(* CODESYS project integratedManufacturingSystem.export

Project tree, tasks and I/O mapping:
  Device : CODESYS Control Win V3 x64, CODESYS, version 3.5.22.30
    application Application
      libraries: Standard, 3.5.22.0 (System)
      task MainTask (cyclic, interval t#20ms, priority 1) calls PLC_PRG
      DUTs/
        data type E_AssemblerState
        data type E_BatchStorageState
        data type E_MachiningCellState
        data type E_PackoutCarrierState
        data type E_PackoutLoaderState
        data type E_PackoutState
        data type E_PairCoordinatorState
        data type E_PairDiverterState
        data type E_PlantState
        data type E_ProductionPhase
        data type E_RackSlotState
        data type E_StorageState
        data type E_TankState
        data type E_TransferState
      GVLs/
        global variables FIO
        global variables PlantConstants
        global variables SCADA
      POUs/
        function block FB_AssemblerCell [ST]
        function block FB_AssemblyUnit [ST]
        function block FB_BatchStorageUnit [ST]
        function block FB_MachiningCell [ST]
        function block FB_MasterOperatorControl [ST]
        function block FB_PackoutCarrierStation [ST]
        function block FB_PackoutLoader [ST]
        function block FB_PairDiverter [ST]
        function block FB_PlantCoordinator [ST]
        function block FB_RackManager [ST]
        function block FB_Storage [ST]
        function block FB_Tank [ST]
        function block FB_TransferCoordinator [ST]
        function block FB_TwinCellUnit [ST]
        function block FB_UnitOperatorControl [ST]
      program PLC_PRG [ST]
      Symbols
*)

// Device/Application/DUTs/E_AssemblerState
{attribute 'qualified_only'}
{attribute 'strict'}
TYPE E_AssemblerState :
(
    Stopped               := 0,
    Homing                := 10,
    WaitingForParts       := 20,
    ClampingParts         := 30,
    LoweringToLid         := 40,
    GrippingLid           := 50,
    ReleasingLidClamp     := 60,
    RaisingLid            := 70,
    MovingToBase          := 80,
    LoweringToBase        := 90,
    ReleasingLid          := 100,
    RaisingFromBase       := 110,
    ReturningHome         := 120,
    ReleasingProduct      := 130,
    WaitingForProductExit := 140,
    Faulted               := 900
);
END_TYPE

// Device/Application/DUTs/E_BatchStorageState
{attribute 'qualified_only'}
{attribute 'strict'}
TYPE E_BatchStorageState :
(
    Stopped                   := 0,
    Idle                      := 10,
    ReservingSlot             := 20,
    WaitingForBatch           := 30,
    DischargingBatch          := 40,
    StoringProduct            := 50,
    CommittingInventory       := 60,
    WaitingForStorageComplete := 70,
    Faulted                   := 900
);
END_TYPE

// Device/Application/DUTs/E_MachiningCellState
{attribute 'qualified_only'}
{attribute 'strict'}
TYPE E_MachiningCellState :
(
    Stopped          := 0,
    Ready            := 10,
    FeedingRaw       := 20,
    WaitingForPickup := 30,
    Processing       := 40,
    Complete         := 50,
    Faulted          := 900
);
END_TYPE

// Device/Application/DUTs/E_PackoutCarrierState
{attribute 'qualified_only'}
{attribute 'strict'}
TYPE E_PackoutCarrierState :
(
    Stopped                      := 0,
    WaitingForCarrierRequest     := 10,
    FeedingCarrier               := 20,
    HoldingCarrierAtLoad         := 30,
    RequestingPlantStorage       := 40,
    TransferringCarrier          := 50,
    WaitingForDownstreamAckClear := 60,
    Faulted                      := 900
);
END_TYPE

// Device/Application/DUTs/E_PackoutLoaderState
{attribute 'qualified_only'}
{attribute 'strict'}
TYPE E_PackoutLoaderState :
(
    Stopped                  := 0,
    Homing                   := 10,
    WaitingForCarrier        := 20,
    WaitingForProduct        := 30,
    MovingToProduct          := 35,
    LoweringToProduct        := 40,
    GrippingProduct          := 50,
    RaisingProduct           := 60,
    MovingToCarrier          := 70,
    LoweringToCarrier        := 80,
    ReleasingProduct         := 90,
    RaisingFromCarrier       := 100,
    ReturningHome            := 110,
    VerifyingLoad            := 120,
    WaitingForLoadAcceptance := 130,
    Complete                 := 140,
    Faulted                  := 900
);
END_TYPE

// Device/Application/DUTs/E_PackoutState
{attribute 'qualified_only'}
{attribute 'strict'}
TYPE E_PackoutState :
(
    Stopped            := 0,
    Homing             := 10,
    WaitingForProduct  := 20,
    RequestingCarrier  := 30,
    PositioningCarrier := 40,
    LoweringToProduct  := 50,
    GrippingProduct    := 60,
    RaisingProduct     := 70,
    MovingToCarrier    := 80,
    LoweringToCarrier  := 90,
    ReleasingProduct   := 100,
    RaisingFromCarrier := 110,
    ReturningHome      := 120,
    VerifyingLoad      := 130,
    ReleasingCarrier   := 140,
    Complete           := 150,
    Faulted            := 900
);
END_TYPE

// Device/Application/DUTs/E_PairCoordinatorState
{attribute 'qualified_only'}
{attribute 'strict'}
TYPE E_PairCoordinatorState :
(
    Stopped          := 0,
    Ready            := 10,
    WaitPairComplete := 20,
    MergeClearance   := 30,
    Faulted          := 900
);
END_TYPE

// Device/Application/DUTs/E_PairDiverterState
{attribute 'qualified_only'}
{attribute 'strict'}
TYPE E_PairDiverterState :
(
    Idle                    := 0,
    ReleasingBase           := 10,
    ReleasingLid            := 20,
    PassingBase             := 30,
    WaitingForLidAtPusher   := 40,
    PositioningLid          := 50,
    PushingLid              := 60,
    WaitingForPartsAtPlace  := 70,
    Complete                := 80,
    Faulted                 := 900
);
END_TYPE

// Device/Application/DUTs/E_PlantState
{attribute 'qualified_only'}
{attribute 'strict'}
TYPE E_PlantState :
(
    Stopped          := 0,
    Ready            := 10,
    Starting         := 20,
    Running          := 30,
    Stopping         := 40,
    Faulted          := 900,
    RecoveryRequired := 910
);
END_TYPE

// Device/Application/DUTs/E_ProductionPhase
{attribute 'qualified_only'}
{attribute 'strict'}
TYPE E_ProductionPhase :
(
    Idle              := 0,
    ReservingStorage  := 10,
    ProducingPair     := 20,
    Assembling        := 30,
    WaitingForPackout := 40,
    Batching          := 50,
    Storing           := 60,
    Complete          := 70
);
END_TYPE

// Device/Application/DUTs/E_RackSlotState
{attribute 'qualified_only'}
{attribute 'strict'}
TYPE E_RackSlotState :
(
    Free     := 0,
    Reserved := 10,
    Occupied := 20,
    Unknown  := 900
);
END_TYPE

// Device/Application/DUTs/E_StorageState
{attribute 'qualified_only'}
{attribute 'strict'}
TYPE E_StorageState :
(
    Stopped                := 0,
    Idle                   := 10,
    ReceivingProduct       := 20,
    ExtendingToLoad        := 30,
    LiftingProduct         := 40,
    RetractingWithProduct  := 50,
    MovingToRack           := 60,
    ExtendingToRack        := 70,
    LoweringProduct        := 80,
    RetractingAfterDeposit := 90,
    ReturningHome          := 100,
    Complete               := 110,
    Faulted                := 900
);
END_TYPE

// Device/Application/DUTs/E_TankState
{attribute 'qualified_only'}
{attribute 'strict'}
TYPE E_TankState :
(
    Stopped     := 0,
    Idle        := 10,
    Filling     := 20,
    BatchReady  := 30,
    Discharging := 40,
    Faulted     := 900
);
END_TYPE

// Device/Application/DUTs/E_TransferState
{attribute 'qualified_only'}
{attribute 'strict'}
TYPE E_TransferState :
(
    Idle                   := 0,
    WaitingForReady        := 10,
    Transferring           := 20,
    WaitingForRequestClear := 30,
    Faulted                := 900
);
END_TYPE

// Device/Application/GVLs/FIO
{attribute 'qualified_only'}
VAR_GLOBAL
    // Factory I/O lifecycle
    rFactoryIOTimeScale : REAL;
    xFactoryIOPaused    : BOOL;
    xFactoryIOReset     : BOOL;
    xFactoryIORunning   : BOOL;
	
	// MASTER operator panel
	xMasterAutoModeSelected       : BOOL;
	xMasterEmergencyStopHealthy   : BOOL;
	xMasterManualModeSelected     : BOOL;
	xMasterResetLightCmd          : BOOL;
	xMasterResetPB                : BOOL;
	xMasterStackGreenCmd          : BOOL;
	xMasterStackRedCmd            : BOOL;
	xMasterStackYellowCmd         : BOOL;
	xMasterStartLightCmd          : BOOL;
	xMasterStartPB                : BOOL;
	xMasterStopCircuitHealthy     : BOOL;
	xMasterStopLightCmd           : BOOL;

    // Plant panel
    xPlantAutoModeSelected     : BOOL;
    xPlantEmergencyStopHealthy : BOOL;
    xPlantManualModeSelected   : BOOL;
    xPlantResetPB              : BOOL;
    xPlantStartPB              : BOOL;
    xPlantStopCircuitHealthy   : BOOL;

    // Twin Cell
    diTwinCellBasesCenterProgress : DINT;
    diTwinCellLidsCenterProgress  : DINT;
    xTwinCellBasesCenterBusy      : BOOL;
    xTwinCellBasesCenterHasError  : BOOL;
    xTwinCellBasesCenterOpened    : BOOL;
    xTwinCellBasesEntryBeamClear  : BOOL;
    xTwinCellBasesExitBeamClear   : BOOL;
    xTwinCellEmergencyStopHealthy : BOOL;
    xTwinCellLidsCenterBusy       : BOOL;
    xTwinCellLidsCenterHasError   : BOOL;
    xTwinCellLidsCenterOpened     : BOOL;
    xTwinCellLidsEntryBeamClear   : BOOL;
    xTwinCellLidsExitBeamClear    : BOOL;
    xTwinCellLocalModeSelected    : BOOL;
    xTwinCellPlantModeSelected    : BOOL;
    xTwinCellResetPB              : BOOL;
    xTwinCellStartPB              : BOOL;
    xTwinCellStopCircuitHealthy   : BOOL;

    // Pair sorter
    xPairSorterCountBeamClear  : BOOL;
    xPairSorterPusherAtBack    : BOOL;
    xPairSorterPusherAtFront   : BOOL;
    xPairSorterPusherBeamClear : BOOL;

    // Assembly
    xAssemblyBaseAtPlace            : BOOL;
    xAssemblyBaseClamped            : BOOL;
    xAssemblyBasesPositionerAtLimit : BOOL;
    xAssemblyItemDetected           : BOOL;
    xAssemblyLidAtPlace             : BOOL;
    xAssemblyLidClamped             : BOOL;
    xAssemblyLidsPositionerAtLimit  : BOOL;
    xAssemblyMovingX                : BOOL;
    xAssemblyMovingZ                : BOOL;
    xAssemblyProductAtOutfeed       : BOOL;

    // Packout
    xPackoutItemDetected           : BOOL;
    xPackoutMovingX                : BOOL;
    xPackoutMovingZ                : BOOL;
    xPackoutPalletAtLoadBeamClear  : BOOL;
    xPackoutProductAtPickBeamClear : BOOL;
    xPackoutProductLoaded          : BOOL;

    // Tank and transfer
    rTankFlowV         : REAL;
    rTankLevelV        : REAL;
    xTankCarrierAtFill : BOOL;
    xTankLevelHighHigh : BOOL;

    // Storage and rack
    xStorageAtEntryBeamClear  : BOOL;
    xStorageAtExitBeamClear   : BOOL;
    xStorageAtUnloadBeamClear : BOOL;
    xStorageForkAtLeft        : BOOL;
    xStorageForkAtMiddle      : BOOL;
    xStorageForkAtRight       : BOOL;
    xStorageLoadBeamClear     : BOOL;
    xStorageMovingX           : BOOL;
    xStorageMovingZ           : BOOL;
	
    // Factory I/O lifecycle — PLC to Factory I/O
    diFactoryIOCameraPositionCmd : DINT;
    xFactoryIOPauseCmd           : BOOL;
    xFactoryIOResetCmd           : BOOL;
    xFactoryIORunCmd             : BOOL;

    // Plant panel — PLC to Factory I/O
    xPlantResetLightCmd : BOOL;
    xPlantStartLightCmd : BOOL;
    xPlantStopLightCmd  : BOOL;

    // Twin Cell — PLC to Factory I/O
    diTwinCellBasesCellCounterDisplay  : DINT;
    diTwinCellBasesPanelCounterDisplay : DINT;
    diTwinCellLidsCellCounterDisplay   : DINT;
    diTwinCellLidsPanelCounterDisplay  : DINT;
    xTwinCellBasesCenterProduceCmd     : BOOL;
    xTwinCellBasesCenterResetCmd       : BOOL;
    xTwinCellBasesCenterStartCmd       : BOOL;
    xTwinCellBasesCenterStopCmd        : BOOL;
    xTwinCellBasesEmitterCmd           : BOOL;
    xTwinCellBasesExitConveyor1Cmd     : BOOL;
    xTwinCellBasesExitConveyor2Cmd     : BOOL;
    xTwinCellBasesRawConveyorCmd       : BOOL;
    xTwinCellLidsCenterProduceCmd      : BOOL;
    xTwinCellLidsCenterResetCmd        : BOOL;
    xTwinCellLidsCenterStartCmd        : BOOL;
    xTwinCellLidsCenterStopCmd         : BOOL;
    xTwinCellLidsEmitterCmd            : BOOL;
    xTwinCellLidsExitConveyor1Cmd      : BOOL;
    xTwinCellLidsExitConveyor2Cmd      : BOOL;
    xTwinCellLidsRawConveyorCmd        : BOOL;
    xTwinCellResetLightCmd             : BOOL;
    xTwinCellStartLightCmd             : BOOL;
    xTwinCellStopLightCmd              : BOOL;

    // Pair sorter — PLC to Factory I/O
    diPairSorterDetectionCountDisplay : DINT;
    xPairSorterBaseCurveConveyorCmd   : BOOL;
    xPairSorterInfeedConveyorCmd      : BOOL;
    xPairSorterPusherCmd              : BOOL;
    xPairSorterPusherZoneConveyorCmd  : BOOL;

    // Assembly — PLC to Factory I/O
    xAssemblyBaseClampCmd            : BOOL;
    xAssemblyBasesConveyorCmd        : BOOL;
    xAssemblyBasesPositionerRaiseCmd : BOOL;
    xAssemblyGrabCmd                 : BOOL;
    xAssemblyLidClampCmd             : BOOL;
    xAssemblyLidsConveyorCmd         : BOOL;
    xAssemblyLidsPositionerRaiseCmd  : BOOL;
    xAssemblyMoveXCmd                : BOOL;
    xAssemblyMoveZCmd                : BOOL;

    // Packout — PLC to Factory I/O
    xPackoutBufferConveyor1Cmd       : BOOL;
    xPackoutBufferConveyor2Cmd       : BOOL;
    xPackoutBufferConveyor3Cmd       : BOOL;
    xPackoutCarrierConveyorCmd       : BOOL;
    xPackoutCarrierEmitterCmd        : BOOL;
    xPackoutCarrierInfeedConveyorCmd : BOOL;
    xPackoutGrabCmd                  : BOOL;
    xPackoutMoveXCmd                 : BOOL;
    xPackoutMoveZCmd                 : BOOL;
    xPackoutPickConveyorCmd          : BOOL;

    // Tank and transfer — PLC to Factory I/O
    rTankDischargeValveCmdV   : REAL;
    rTankFillValveCmdV        : REAL;
    xTankTransferConveyor1Cmd : BOOL;
    xTankTransferConveyor2Cmd : BOOL;
    xTankTransferConveyor3Cmd : BOOL;
    xTankTransferConveyor4Cmd : BOOL;

    // Storage and rack — PLC to Factory I/O
    wStorageTargetPositionCmd : WORD := 55;
    xStorageEntryConveyorCmd  : BOOL;
    xStorageExitConveyorCmd   : BOOL;
    xStorageExitRemoverCmd    : BOOL;
    xStorageForksLeftCmd      : BOOL;
    xStorageForksRightCmd     : BOOL;
    xStorageLiftCmd           : BOOL;
    xStorageLoadConveyorCmd   : BOOL;
    xStorageUnloadConveyorCmd : BOOL;

    // Stack lights — PLC to Factory I/O
    xPackoutStackGreenCmd  : BOOL;
    xPackoutStackRedCmd    : BOOL;
    xPackoutStackYellowCmd : BOOL;
    xPlantStackGreenCmd    : BOOL;
    xPlantStackRedCmd      : BOOL;
    xPlantStackYellowCmd   : BOOL;
    xStorageStackGreenCmd  : BOOL;
    xStorageStackRedCmd    : BOOL;
    xStorageStackYellowCmd : BOOL;
    xTankStackGreenCmd     : BOOL;
    xTankStackRedCmd       : BOOL;
    xTankStackYellowCmd    : BOOL;
END_VAR

// Device/Application/GVLs/PlantConstants
{attribute 'qualified_only'}
VAR_GLOBAL CONSTANT
    tPairTransferTimeout    : TIME := T#2M;
    tProductTransferTimeout : TIME := T#30S;
    wStorageHomePosition    : WORD := 55;
END_VAR

// Device/Application/GVLs/SCADA
{attribute 'symbol' := 'read'}
{attribute 'qualified_only'}
VAR_GLOBAL
    // Ignition to PLC — momentary requests
	 {attribute 'symbol' := 'readwrite'}
    xResetReq : BOOL;
	 {attribute 'symbol' := 'readwrite'}
    xStartReq : BOOL;
	 {attribute 'symbol' := 'readwrite'}
    xStopReq  : BOOL;
	 {attribute 'symbol' := 'readwrite'}
	xAutoModeSelected 		  : BOOL := FALSE;

    // PLC to Ignition — plant
    diPlantCompletedLoadCount : DINT;
    ePlantState               : E_PlantState := E_PlantState.Stopped;
    eProductionPhase          : E_ProductionPhase := E_ProductionPhase.Idle;
    uiPlantFaultCode          : UINT;
	xAllEmergencyStopsHealthy : BOOL;
	xAutoModeActive           : BOOL;
	xFactoryIORunning         : BOOL;
	xManualModeActive         : BOOL;
    xPlantFaulted             : BOOL;
    xPlantRecoveryRequired    : BOOL;
    xPlantRunning             : BOOL;
    xPlantStopPending         : BOOL;

    // PLC to Ignition — Twin Cell
    diTwinCellPairCount : DINT;
    uiTwinCellFaultCode : UINT;
    xTwinCellBusy       : BOOL;
    xTwinCellFaulted    : BOOL;
    xTwinCellReady      : BOOL;

    // PLC to Ignition — pair transfer
    ePairTransferState       : E_TransferState := E_TransferState.Idle;
    uiPairTransferFaultCode  : UINT;
    xPairTransferAck         : BOOL;
    xPairTransferFaulted     : BOOL;
    xPairTransferPermit      : BOOL;
    xPairTransferReady       : BOOL;
    xPairTransferReq         : BOOL;

    // PLC to Ignition — pair sorter
    diPairSorterDetectionCount : DINT;
    ePairDiverterState         : E_PairDiverterState := E_PairDiverterState.Idle;
    uiPairSorterFaultCode      : UINT;
    xPairSorterFaulted         : BOOL;
    xPairSorterPartAtPusher    : BOOL;

    // PLC to Ignition — assembly
    diAssemblyProductCount : DINT;
    eAssemblyState         : E_AssemblerState := E_AssemblerState.Stopped;
    uiAssemblyFaultCode    : UINT;
    xAssemblyBusy          : BOOL;
    xAssemblyFaulted       : BOOL;
    xAssemblyReady         : BOOL;

    // PLC to Ignition — product transfer
    eProductTransferState      : E_TransferState := E_TransferState.Idle;
    uiProductTransferFaultCode : UINT;
    xProductTransferAck        : BOOL;
    xProductTransferFaulted    : BOOL;
    xProductTransferPermit     : BOOL;
    xProductTransferReady      : BOOL;
    xProductTransferReq        : BOOL;

    // PLC to Ignition — packout
	diPackoutProductCount        : DINT;
	
	ePackoutCarrierState         : E_PackoutCarrierState :=
									   E_PackoutCarrierState.Stopped;
	ePackoutLoaderState          : E_PackoutLoaderState :=
									   E_PackoutLoaderState.Stopped;
	
	uiPackoutCarrierFaultCode    : UINT;
	uiPackoutLoaderFaultCode     : UINT;
	
	xPackoutBusy                 : BOOL;
	xPackoutCarrierBusy          : BOOL;
	xPackoutCarrierFaulted       : BOOL;
	xPackoutCarrierReady         : BOOL;
	xPackoutFaulted              : BOOL;
	xPackoutLoaderBusy           : BOOL;
	xPackoutLoaderFaulted        : BOOL;
	xPackoutLoaderReady          : BOOL;
	xPackoutReady                : BOOL;

    // PLC to Ignition — process and storage
    eBatchStorageState       : E_BatchStorageState := E_BatchStorageState.Stopped;
    eStorageState            : E_StorageState := E_StorageState.Stopped;
    eTankState               : E_TankState := E_TankState.Stopped;
    rTankLevelPct            : REAL;
    uiRackFreeCount          : UINT;
    uiRackOccupiedCount      : UINT;
    uiRackReservedCount      : UINT;
    uiRackUnknownCount       : UINT;
    uiStorageFaultCode       : UINT;
    wStorageReservedPosition : WORD;
    xPackoutPalletAtLoad     : BOOL;
    xPackoutProductAtPick    : BOOL;
    xPackoutProductLoaded    : BOOL;
    xRackFull                : BOOL;
    xStorageBusy             : BOOL;
    xStorageFaulted          : BOOL;
    xStorageReady            : BOOL;
	
	// Maintained automatic-mode request from Ignition.
	{attribute 'symbol' := 'readwrite'}
	xIgnitionAutoModeReq : BOOL;
END_VAR

// Device/Application/PLC_PRG
PROGRAM PLC_PRG
VAR
    // Function-block instances
	fbAssemblyUnit                  : FB_AssemblyUnit;
	fbBatchStorageOperatorControl   : FB_UnitOperatorControl;
	fbBatchStorageUnit              : FB_BatchStorageUnit;
	fbMasterOperatorControl         : FB_MasterOperatorControl;
	fbPackoutCarrierStation         : FB_PackoutCarrierStation;
	fbPackoutLoader                 : FB_PackoutLoader;
	fbPairDiverter                  : FB_PairDiverter;
	fbPairTransfer                  : FB_TransferCoordinator;
	fbPlantCoordinator              : FB_PlantCoordinator;
	fbProductTransfer               : FB_TransferCoordinator;
	fbTwinCellOperatorControl       : FB_UnitOperatorControl;
	fbTwinCellUnit                  : FB_TwinCellUnit;

    // Normalised physical inputs
    rTankLevelPct               : REAL;
	xBatchStorageTransferActive : BOOL;
    xPackoutPalletAtLoad        : BOOL;
    xPackoutProductAtPick       : BOOL;
    xPairSorterCountDetected    : BOOL;
    xPairSorterPartAtPusher     : BOOL;
    xStorageAtEntry             : BOOL;
    xStorageAtExit              : BOOL;
    xStorageAtUnload            : BOOL;
	xStorageCraneAtHome         : BOOL;
    xStorageProductAtLoad       : BOOL;
    xTwinCellBasesEntryDetected : BOOL;
    xTwinCellBasesExitDetected  : BOOL;
    xTwinCellLidsEntryDetected  : BOOL;
    xTwinCellLidsExitDetected   : BOOL;
	xTwinCellOutputPermit 		: BOOL := TRUE;

    // Safety and commissioning
    xAllEmergencyStopsHealthy : BOOL;
	xAnyFault              	  : BOOL;
	xOutputPermit             : BOOL;
	xPairSorterOutputPermit   : BOOL := TRUE;
    xPairTransferActive    	  : BOOL;
    xProductTransferActive    : BOOL;
	xStorageOutputPermit      : BOOL;
END_VAR

// =============================================================
// 1. INPUT IMAGE AND POLARITY NORMALISATION
// =============================================================
rTankLevelPct := FIO.rTankLevelV * 10.0;

xPackoutPalletAtLoad := NOT FIO.xPackoutPalletAtLoadBeamClear;
xPackoutProductAtPick := NOT FIO.xPackoutProductAtPickBeamClear;
xPairSorterCountDetected := NOT FIO.xPairSorterCountBeamClear;
xPairSorterPartAtPusher := NOT FIO.xPairSorterPusherBeamClear;

xStorageAtEntry := NOT FIO.xStorageAtEntryBeamClear;
xStorageAtExit := NOT FIO.xStorageAtExitBeamClear;
xStorageAtUnload := NOT FIO.xStorageAtUnloadBeamClear;
xStorageCraneAtHome :=
    (FIO.wStorageTargetPositionCmd =
        PlantConstants.wStorageHomePosition)
    AND FIO.xStorageForkAtMiddle
    AND NOT FIO.xStorageMovingX
    AND NOT FIO.xStorageMovingZ;
xStorageProductAtLoad := NOT FIO.xStorageLoadBeamClear;

xTwinCellBasesEntryDetected := NOT FIO.xTwinCellBasesEntryBeamClear;
xTwinCellBasesExitDetected := NOT FIO.xTwinCellBasesExitBeamClear;
xTwinCellLidsEntryDetected := NOT FIO.xTwinCellLidsEntryBeamClear;
xTwinCellLidsExitDetected := NOT FIO.xTwinCellLidsExitBeamClear;

// =============================================================
// 2. SAFETY AND COMMISSIONING CONDITIONS
// =============================================================
xAllEmergencyStopsHealthy :=
    FIO.xMasterEmergencyStopHealthy
	AND FIO.xPlantEmergencyStopHealthy
    AND FIO.xTwinCellEmergencyStopHealthy;

// Global commissioned outputs are permitted.
// Uncommissioned zones remain protected by their individual permits.
xOutputPermit := TRUE;

// =============================================================
// 3. OPERATOR CONTROL
// =============================================================
fbMasterOperatorControl(
    xAutoModeSelected :=
		FIO.xMasterAutoModeSelected
		OR SCADA.xIgnitionAutoModeReq,
    xEmergencyStopHealthy := xAllEmergencyStopsHealthy,
    xFactoryIORunning := FIO.xFactoryIORunning,
    xManualModeSelected := FIO.xMasterManualModeSelected,
    xPlantFaulted := fbPlantCoordinator.xFaulted,
    xResetPB := FIO.xMasterResetPB OR SCADA.xResetReq,
    xStartPB := FIO.xMasterStartPB OR SCADA.xStartReq,
    xStopCircuitHealthy :=
        FIO.xMasterStopCircuitHealthy
        AND NOT SCADA.xStopReq
);

xBatchStorageTransferActive :=
    fbBatchStorageUnit.xBusy
    OR fbPackoutCarrierStation.xBusy
    OR fbPackoutCarrierStation.xLoadedCarrierReq
    OR fbPackoutLoader.xBusy
    OR fbPackoutLoader.xLoadComplete;

fbBatchStorageOperatorControl(
    xEmergencyStopHealthy := xAllEmergencyStopsHealthy,
    xLocalModeSelected := FIO.xPlantManualModeSelected,
    xLocalResetPB := FIO.xPlantResetPB,
    xLocalStartPB := FIO.xPlantStartPB,
    xLocalStopHealthy := FIO.xPlantStopCircuitHealthy,
    xMasterAutoModeActive :=
        fbMasterOperatorControl.xAutoModeActive,
    xMasterEnable := fbMasterOperatorControl.xEnable,
    xMasterManualModeActive :=
        fbMasterOperatorControl.xManualModeActive,
    xMasterModeSelected := FIO.xPlantAutoModeSelected,
    xMasterResetPulse := fbMasterOperatorControl.xResetPulse,
    xMasterRun := fbPlantCoordinator.xRunning,
    xTransferActive := xBatchStorageTransferActive
);

xPairTransferActive :=
    fbPairTransfer.eState <> E_TransferState.Idle;

xProductTransferActive :=
    (fbProductTransfer.eState <> E_TransferState.Idle)
    OR fbPackoutLoader.xBusy
    OR fbPackoutLoader.xLoadComplete;

fbTwinCellOperatorControl(
    xEmergencyStopHealthy := xAllEmergencyStopsHealthy,
    xLocalModeSelected := FIO.xTwinCellLocalModeSelected,
    xLocalResetPB := FIO.xTwinCellResetPB,
    xLocalStartPB := FIO.xTwinCellStartPB,
    xLocalStopHealthy := FIO.xTwinCellStopCircuitHealthy,
	xMasterAutoModeActive :=
    	fbMasterOperatorControl.xAutoModeActive,
    xMasterEnable := fbMasterOperatorControl.xEnable,
	xMasterManualModeActive :=
    	fbMasterOperatorControl.xManualModeActive,
    xMasterModeSelected := FIO.xTwinCellPlantModeSelected,
    xMasterResetPulse := fbMasterOperatorControl.xResetPulse,
    xMasterRun := fbPlantCoordinator.xRunning,
    xTransferActive :=
        xPairTransferActive OR xProductTransferActive
);

// =============================================================
// 4. UNIT BOUNDARIES
// =============================================================
fbTwinCellUnit(
    xEnable := fbTwinCellOperatorControl.xEnable,
    xPairAccepted := fbAssemblyUnit.xPairAck,
	xProductionRequest :=
		fbMasterOperatorControl.xAutoRun
		AND fbPlantCoordinator.xAllowNewPair,
    xReset := fbTwinCellOperatorControl.xResetPulse,
    xRun :=
		fbTwinCellOperatorControl.xRun
		AND xTwinCellOutputPermit,
    xTwinCellBasesCenterBusy :=
        FIO.xTwinCellBasesCenterBusy,
    xTwinCellBasesCenterHasError :=
        FIO.xTwinCellBasesCenterHasError,
    xTwinCellBasesCenterOpened :=
        FIO.xTwinCellBasesCenterOpened,
    xTwinCellBasesEntryDetected :=
        xTwinCellBasesEntryDetected,
    xTwinCellBasesExitDetected :=
        xTwinCellBasesExitDetected,
    xTwinCellLidsCenterBusy :=
        FIO.xTwinCellLidsCenterBusy,
    xTwinCellLidsCenterHasError :=
        FIO.xTwinCellLidsCenterHasError,
    xTwinCellLidsCenterOpened :=
        FIO.xTwinCellLidsCenterOpened,
    xTwinCellLidsEntryDetected :=
        xTwinCellLidsEntryDetected,
    xTwinCellLidsExitDetected :=
        xTwinCellLidsExitDetected
);

fbAssemblyUnit(
    xBaseAtPlace :=
        FIO.xAssemblyBaseAtPlace,

    xBaseClamped :=
        FIO.xAssemblyBaseClamped,

    xBasesPositionerAtLimit :=
        FIO.xAssemblyBasesPositionerAtLimit,

    xEnable :=
        fbTwinCellOperatorControl.xEnable
        AND FIO.xFactoryIORunning
        AND xOutputPermit,

    xItemDetected :=
        FIO.xAssemblyItemDetected,

    xLidAtPlace :=
        FIO.xAssemblyLidAtPlace,

    xLidClamped :=
        FIO.xAssemblyLidClamped,

    xMovingX :=
        FIO.xAssemblyMovingX,

    xMovingZ :=
        FIO.xAssemblyMovingZ,

    xProductAtOutfeed :=
        FIO.xAssemblyProductAtOutfeed,

    xProductTransferAck :=
        fbPackoutLoader.xProductTransferAck,

    xReset :=
        fbTwinCellOperatorControl.xResetPulse,

    xRun :=
        fbTwinCellOperatorControl.xRun
);

// =============================================================
// 5. P10-TO-P11 TRANSFER
// =============================================================
fbPairTransfer(
    tTransferTimeout := PlantConstants.tPairTransferTimeout,
    xAck := fbAssemblyUnit.xPairAck,
    xEnable :=
		fbPlantCoordinator.xPairTransferEnable
		AND xPairSorterOutputPermit,
    xReady := fbAssemblyUnit.xPairReady,
    xReq := fbTwinCellUnit.xPairReq,
    xReset := fbMasterOperatorControl.xResetPulse,
	xRun := fbTwinCellOperatorControl.xRun
);

fbPairDiverter(
	tLidPositionTime := T#700MS,
    tStepTimeout := T#45S,
    xAssemblyBaseAtPlace := FIO.xAssemblyBaseAtPlace,
    xAssemblyLidAtPlace := FIO.xAssemblyLidAtPlace,
    xCountDetected := xPairSorterCountDetected,
    xEnable :=
		xAllEmergencyStopsHealthy
		AND FIO.xFactoryIORunning
		AND xOutputPermit
		AND xPairSorterOutputPermit,
		xPartAtPusher := xPairSorterPartAtPusher,
    xPusherAtBack := FIO.xPairSorterPusherAtBack,
    xPusherAtFront := FIO.xPairSorterPusherAtFront,
    xReset := fbMasterOperatorControl.xResetPulse,
	xRun := fbTwinCellOperatorControl.xRun,
	xTransferPermit := fbPairTransfer.xPermit
);

// =============================================================
// 6. P11-TO-PACKOUT LOADER TRANSFER
// =============================================================
fbProductTransfer(
    tTransferTimeout := PlantConstants.tProductTransferTimeout,
    xAck := fbPackoutLoader.xProductTransferAck,
    xEnable := fbPlantCoordinator.xProductTransferEnable,
    xReady := fbPackoutLoader.xProductTransferReady,
    xReq := fbAssemblyUnit.xProductReq,
    xReset := fbMasterOperatorControl.xResetPulse,
	xRun := fbTwinCellOperatorControl.xRun	
);

fbPackoutLoader(
    tStepTimeout := T#20S,
    xCarrierReady := fbPackoutCarrierStation.xCarrierReady,
    xEnable :=
        xAllEmergencyStopsHealthy
		AND FIO.xFactoryIORunning
		AND xOutputPermit,
    xItemDetected := FIO.xPackoutItemDetected,
    xLoadAccepted := fbPackoutCarrierStation.xLoadAccepted,
    xMovingX := FIO.xPackoutMovingX,
    xMovingZ := FIO.xPackoutMovingZ,
    xProductAtPick := xPackoutProductAtPick,
    xProductLoaded := FIO.xPackoutProductLoaded,
    xProductTransferPermit := fbProductTransfer.xPermit,
    xReset := fbTwinCellOperatorControl.xResetPulse,
	xRun :=
		fbTwinCellOperatorControl.xRun
		AND fbPlantCoordinator.xRunning
);

fbPackoutCarrierStation(
    tStepTimeout := T#30S,
    xCarrierReq := fbPackoutLoader.xCarrierReq,
    xDownstreamAck := fbBatchStorageUnit.xProductTransferAck,
    xDownstreamReady := fbBatchStorageUnit.xProductTransferReady,
    xEnable :=
        fbBatchStorageOperatorControl.xEnable
        AND FIO.xFactoryIORunning
        AND xOutputPermit,
    xLoadComplete := fbPackoutLoader.xLoadComplete,
    xPalletAtLoad := xPackoutPalletAtLoad,
    xProductLoaded := FIO.xPackoutProductLoaded,
    xReset := fbBatchStorageOperatorControl.xResetPulse,
    xRun :=
        fbBatchStorageOperatorControl.xRun
        AND fbPlantCoordinator.xRunning
);

// =============================================================
// 7. PACKOUT-TO-PLANT STORAGE BOUNDARY
// =============================================================
fbBatchStorageUnit(
    rTankLevelV := FIO.rTankLevelV,
	wStorageHomePosition :=
        PlantConstants.wStorageHomePosition,
    xEnable := fbBatchStorageOperatorControl.xEnable,
    xPackoutPalletAtLoad := xPackoutPalletAtLoad,
    xPackoutProductLoaded := FIO.xPackoutProductLoaded,
    xProductTransferReq :=
        fbPackoutCarrierStation.xLoadedCarrierReq,
    xReset := fbBatchStorageOperatorControl.xResetPulse,
    xRun := fbBatchStorageOperatorControl.xRun,
    xStorageAtEntry := xStorageAtEntry,
	 xStorageCraneAtHome := xStorageCraneAtHome,
    xStorageForkAtLeft := FIO.xStorageForkAtLeft,
    xStorageForkAtMiddle := FIO.xStorageForkAtMiddle,
    xStorageForkAtRight := FIO.xStorageForkAtRight,
    xStorageMovingX := FIO.xStorageMovingX,
    xStorageMovingZ := FIO.xStorageMovingZ,
    xStorageProductAtLoad := xStorageProductAtLoad,
    xTankCarrierAtFill := FIO.xTankCarrierAtFill,
    xTankLevelHighHigh := FIO.xTankLevelHighHigh
);

// =============================================================
// 8. PLANT COORDINATION
// =============================================================
xAnyFault :=
    fbAssemblyUnit.xFaulted
    OR fbBatchStorageUnit.xFaulted
    OR fbPackoutCarrierStation.xFaulted
    OR fbPackoutLoader.xFaulted
    OR fbPairDiverter.xFaulted
    OR fbPairTransfer.xFaulted
    OR fbProductTransfer.xFaulted
    OR fbTwinCellUnit.xFaulted;

fbPlantCoordinator(
    xAnyFault := xAnyFault,
    xAutoRun := fbMasterOperatorControl.xAutoRun,
    xBatchStorageReady := fbBatchStorageUnit.xReady,
    xEnable := fbMasterOperatorControl.xEnable,
    xPairTransferComplete := fbPairTransfer.xComplete,
    xProductTransferComplete := fbProductTransfer.xComplete,
    xRackCommitAck := fbBatchStorageUnit.xRackCommitAck,
    xRackReservationValid := fbBatchStorageUnit.xRackReservationValid,
    xReset := fbMasterOperatorControl.xResetPulse
);

// Consume momentary SCADA requests after the FBs have sampled them.
SCADA.xResetReq := FALSE;
SCADA.xStartReq := FALSE;
SCADA.xStopReq := FALSE;

// =============================================================
// 9. SCADA STATUS PUBLICATION
// =============================================================

// Plant
SCADA.diPlantCompletedLoadCount :=
    UINT_TO_DINT(fbBatchStorageUnit.uiRackOccupiedCount);

SCADA.ePlantState :=
    fbPlantCoordinator.eState;

SCADA.eProductionPhase :=
    fbPlantCoordinator.eProductionPhase;

SCADA.uiPlantFaultCode :=
    fbPlantCoordinator.uiFaultCode;

SCADA.xAllEmergencyStopsHealthy :=
    xAllEmergencyStopsHealthy;

SCADA.xAutoModeActive :=
    fbMasterOperatorControl.xAutoModeActive;

SCADA.xFactoryIORunning :=
    FIO.xFactoryIORunning;

SCADA.xManualModeActive :=
    fbMasterOperatorControl.xManualModeActive;

SCADA.xPlantFaulted :=
    fbPlantCoordinator.xFaulted;

SCADA.xPlantRecoveryRequired :=
    fbPlantCoordinator.xRecoveryRequired;

SCADA.xPlantRunning :=
    fbPlantCoordinator.xRunning;

SCADA.xPlantStopPending :=
    fbPlantCoordinator.xStopPending;


// Twin Cell
SCADA.diTwinCellPairCount :=
    fbTwinCellUnit.diPairCount;

SCADA.uiTwinCellFaultCode :=
    fbTwinCellUnit.uiFaultCode;

SCADA.xTwinCellBusy :=
    fbTwinCellUnit.xBusy;

SCADA.xTwinCellFaulted :=
    fbTwinCellUnit.xFaulted;

SCADA.xTwinCellReady :=
    fbTwinCellUnit.xReady;


// Pair transfer
SCADA.ePairTransferState :=
    fbPairTransfer.eState;

SCADA.uiPairTransferFaultCode :=
    fbPairTransfer.uiFaultCode;

SCADA.xPairTransferAck :=
    fbAssemblyUnit.xPairAck;

SCADA.xPairTransferFaulted :=
    fbPairTransfer.xFaulted;

SCADA.xPairTransferPermit :=
    fbPairTransfer.xPermit;

SCADA.xPairTransferReady :=
    fbAssemblyUnit.xPairReady;

SCADA.xPairTransferReq :=
    fbTwinCellUnit.xPairReq;


// Pair sorter
SCADA.diPairSorterDetectionCount :=
    fbPairDiverter.diDetectionCount;

SCADA.ePairDiverterState :=
    fbPairDiverter.eState;

SCADA.uiPairSorterFaultCode :=
    fbPairDiverter.uiFaultCode;

SCADA.xPairSorterFaulted :=
    fbPairDiverter.xFaulted;

SCADA.xPairSorterPartAtPusher :=
    xPairSorterPartAtPusher;


// Assembly
SCADA.diAssemblyProductCount :=
    fbAssemblyUnit.diProductCount;

SCADA.eAssemblyState :=
    fbAssemblyUnit.eState;

SCADA.uiAssemblyFaultCode :=
    fbAssemblyUnit.uiFaultCode;

SCADA.xAssemblyBusy :=
    fbAssemblyUnit.xBusy;

SCADA.xAssemblyFaulted :=
    fbAssemblyUnit.xFaulted;

SCADA.xAssemblyReady :=
    fbAssemblyUnit.xReady;


// Product transfer
SCADA.eProductTransferState :=
    fbProductTransfer.eState;

SCADA.uiProductTransferFaultCode :=
    fbProductTransfer.uiFaultCode;

SCADA.xProductTransferAck :=
    fbPackoutLoader.xProductTransferAck;

SCADA.xProductTransferFaulted :=
    fbProductTransfer.xFaulted;

SCADA.xProductTransferPermit :=
    fbProductTransfer.xPermit;

SCADA.xProductTransferReady :=
    fbPackoutLoader.xProductTransferReady;

SCADA.xProductTransferReq :=
    fbAssemblyUnit.xProductReq;


// Packout
SCADA.diPackoutProductCount :=
    fbPackoutLoader.diProductCount;

SCADA.ePackoutCarrierState :=
    fbPackoutCarrierStation.eState;

SCADA.ePackoutLoaderState :=
    fbPackoutLoader.eState;

SCADA.uiPackoutCarrierFaultCode :=
    fbPackoutCarrierStation.uiFaultCode;

SCADA.uiPackoutLoaderFaultCode :=
    fbPackoutLoader.uiFaultCode;

SCADA.xPackoutBusy :=
    fbPackoutCarrierStation.xBusy
    OR fbPackoutLoader.xBusy;

SCADA.xPackoutCarrierBusy :=
    fbPackoutCarrierStation.xBusy;

SCADA.xPackoutCarrierFaulted :=
    fbPackoutCarrierStation.xFaulted;

SCADA.xPackoutCarrierReady :=
    fbPackoutCarrierStation.xReady;

SCADA.xPackoutFaulted :=
    fbPackoutCarrierStation.xFaulted
    OR fbPackoutLoader.xFaulted;

SCADA.xPackoutLoaderBusy :=
    fbPackoutLoader.xBusy;

SCADA.xPackoutLoaderFaulted :=
    fbPackoutLoader.xFaulted;

SCADA.xPackoutLoaderReady :=
    fbPackoutLoader.xReady;

SCADA.xPackoutReady :=
    fbPackoutCarrierStation.xReady
    AND fbPackoutLoader.xReady;


// Plant Storage
SCADA.eBatchStorageState :=
    fbBatchStorageUnit.eState;

SCADA.eStorageState :=
    fbBatchStorageUnit.eStorageState;

SCADA.eTankState :=
    fbBatchStorageUnit.eTankState;

SCADA.rTankLevelPct :=
    rTankLevelPct;

SCADA.uiRackFreeCount :=
    fbBatchStorageUnit.uiRackFreeCount;

SCADA.uiRackOccupiedCount :=
    fbBatchStorageUnit.uiRackOccupiedCount;

SCADA.uiRackReservedCount :=
    fbBatchStorageUnit.uiRackReservedCount;

SCADA.uiRackUnknownCount :=
    fbBatchStorageUnit.uiRackUnknownCount;

SCADA.uiStorageFaultCode :=
    fbBatchStorageUnit.uiStorageFaultCode;

SCADA.wStorageReservedPosition :=
    fbBatchStorageUnit.wRackReservedPosition;

SCADA.xPackoutPalletAtLoad :=
    xPackoutPalletAtLoad;

SCADA.xPackoutProductAtPick :=
    xPackoutProductAtPick;

SCADA.xPackoutProductLoaded :=
    FIO.xPackoutProductLoaded;

SCADA.xRackFull :=
    fbBatchStorageUnit.xRackFull;

SCADA.xStorageBusy :=
    fbBatchStorageUnit.xStorageBusy;

SCADA.xStorageFaulted :=
    fbBatchStorageUnit.xStorageFaulted;

SCADA.xStorageReady :=
    fbBatchStorageUnit.xStorageReady;
	
// =============================================================
// 10. SAFE FIO OUTPUT BOUNDARY — PART 1
// =============================================================

// Factory I/O lifecycle
FIO.diFactoryIOCameraPositionCmd := 0;
FIO.xFactoryIOPauseCmd := FALSE;
FIO.xFactoryIOResetCmd := FALSE;
FIO.xFactoryIORunCmd := FALSE;

// Twin Cell production-count displays
FIO.diTwinCellBasesCellCounterDisplay :=
    fbTwinCellUnit.diBasesCount;

FIO.diTwinCellBasesPanelCounterDisplay :=
    fbTwinCellUnit.diBasesCount;

FIO.diTwinCellLidsCellCounterDisplay :=
    fbTwinCellUnit.diLidsCount;

FIO.diTwinCellLidsPanelCounterDisplay :=
    fbTwinCellUnit.diLidsCount;

// MASTER operator-panel indication
FIO.xMasterResetLightCmd :=
    fbMasterOperatorControl.xResetRequired;

FIO.xMasterStackGreenCmd :=
    xAllEmergencyStopsHealthy
    AND NOT fbPlantCoordinator.xFaulted
    AND fbMasterOperatorControl.xAutoRun;

FIO.xMasterStackRedCmd :=
    NOT xAllEmergencyStopsHealthy
    OR fbPlantCoordinator.xFaulted;

FIO.xMasterStackYellowCmd :=
    xAllEmergencyStopsHealthy
    AND NOT fbPlantCoordinator.xFaulted
    AND NOT fbMasterOperatorControl.xAutoRun;

FIO.xMasterStartLightCmd :=
    fbMasterOperatorControl.xAutoRun;

FIO.xMasterStopLightCmd :=
    NOT fbMasterOperatorControl.xAutoRun;

// Twin Cell panel indication
FIO.xTwinCellResetLightCmd := FALSE;
FIO.xTwinCellStartLightCmd := FALSE;
FIO.xTwinCellStopLightCmd := TRUE;

// Twin Cell — bases
FIO.xTwinCellBasesCenterProduceCmd :=
    xOutputPermit
    AND xTwinCellOutputPermit
    AND fbTwinCellUnit.xBasesCenterProduceCmd;

FIO.xTwinCellBasesCenterResetCmd :=
    xOutputPermit
    AND xTwinCellOutputPermit
    AND fbTwinCellUnit.xBasesCenterResetCmd;

FIO.xTwinCellBasesCenterStartCmd :=
    xOutputPermit
    AND xTwinCellOutputPermit
    AND fbTwinCellUnit.xBasesCenterStartCmd;

FIO.xTwinCellBasesCenterStopCmd :=
    xOutputPermit
    AND xTwinCellOutputPermit
    AND fbTwinCellUnit.xBasesCenterStopCmd;

FIO.xTwinCellBasesEmitterCmd :=
    xOutputPermit
    AND xTwinCellOutputPermit
    AND fbTwinCellUnit.xBasesEmitterCmd;

FIO.xTwinCellBasesExitConveyor1Cmd :=
    xOutputPermit
    AND xTwinCellOutputPermit
    AND (
        fbTwinCellUnit.xBasesExitConveyor1Cmd
        OR (
            xPairSorterOutputPermit
            AND fbPairDiverter.xBasesOutfeedCmd
        )
    );

FIO.xTwinCellBasesExitConveyor2Cmd :=
    xOutputPermit
    AND xTwinCellOutputPermit
    AND (
        fbTwinCellUnit.xBasesExitConveyor2Cmd
        OR (
            xPairSorterOutputPermit
            AND fbPairDiverter.xBasesOutfeedCmd
        )
    );

FIO.xTwinCellBasesRawConveyorCmd :=
    xOutputPermit
    AND xTwinCellOutputPermit
    AND fbTwinCellUnit.xBasesRawConveyorCmd;

// Twin Cell — lids
FIO.xTwinCellLidsCenterProduceCmd :=
    xOutputPermit
    AND xTwinCellOutputPermit
    AND fbTwinCellUnit.xLidsCenterProduceCmd;

FIO.xTwinCellLidsCenterResetCmd :=
    xOutputPermit
    AND xTwinCellOutputPermit
    AND fbTwinCellUnit.xLidsCenterResetCmd;

FIO.xTwinCellLidsCenterStartCmd :=
    xOutputPermit
    AND xTwinCellOutputPermit
    AND fbTwinCellUnit.xLidsCenterStartCmd;

FIO.xTwinCellLidsCenterStopCmd :=
    xOutputPermit
    AND xTwinCellOutputPermit
    AND fbTwinCellUnit.xLidsCenterStopCmd;

FIO.xTwinCellLidsEmitterCmd :=
    xOutputPermit
    AND xTwinCellOutputPermit
    AND fbTwinCellUnit.xLidsEmitterCmd;

FIO.xTwinCellLidsExitConveyor1Cmd :=
    xOutputPermit
    AND xTwinCellOutputPermit
    AND (
        fbTwinCellUnit.xLidsExitConveyor1Cmd
        OR (
            xPairSorterOutputPermit
            AND fbPairDiverter.xLidsOutfeedCmd
        )
    );

FIO.xTwinCellLidsExitConveyor2Cmd :=
    xOutputPermit
    AND xTwinCellOutputPermit
    AND (
        fbTwinCellUnit.xLidsExitConveyor2Cmd
        OR (
            xPairSorterOutputPermit
            AND fbPairDiverter.xLidsOutfeedCmd
        )
    );

FIO.xTwinCellLidsRawConveyorCmd :=
    xOutputPermit
    AND xTwinCellOutputPermit
    AND fbTwinCellUnit.xLidsRawConveyorCmd;

// Pair sorter
FIO.diPairSorterDetectionCountDisplay :=
    fbPairDiverter.diDetectionCount;

FIO.xPairSorterBaseCurveConveyorCmd :=
    xOutputPermit
    AND xPairSorterOutputPermit
    AND fbPairDiverter.xBaseCurveConveyorCmd;

FIO.xPairSorterInfeedConveyorCmd :=
    xOutputPermit
    AND xPairSorterOutputPermit
    AND fbPairDiverter.xInfeedConveyorCmd;

FIO.xPairSorterPusherCmd :=
    xOutputPermit
    AND xPairSorterOutputPermit
    AND fbPairDiverter.xPusherCmd;

FIO.xPairSorterPusherZoneConveyorCmd :=
    xOutputPermit
    AND xPairSorterOutputPermit
    AND fbPairDiverter.xPusherZoneConveyorCmd;

// Assembly
FIO.xAssemblyBaseClampCmd :=
    xOutputPermit
    AND fbTwinCellOperatorControl.xRun
    AND fbAssemblyUnit.xBaseClampCmd;

FIO.xAssemblyBasesConveyorCmd :=
    xOutputPermit
    AND fbTwinCellOperatorControl.xRun
    AND (
        fbAssemblyUnit.xBasesConveyorCmd
        OR (
            xPairSorterOutputPermit
            AND fbPairDiverter.xBasesOutfeedCmd
        )
    );

FIO.xAssemblyBasesPositionerRaiseCmd :=
    xOutputPermit
    AND fbTwinCellOperatorControl.xRun
    AND fbAssemblyUnit.xBasesPositionerRaiseCmd;

FIO.xAssemblyGrabCmd :=
    xOutputPermit
    AND fbTwinCellOperatorControl.xRun
    AND fbAssemblyUnit.xGrabCmd;

FIO.xAssemblyLidClampCmd :=
    xOutputPermit
    AND fbTwinCellOperatorControl.xRun
    AND fbAssemblyUnit.xLidClampCmd;

FIO.xAssemblyLidsConveyorCmd :=
    xOutputPermit
    AND fbTwinCellOperatorControl.xRun
    AND (
        fbAssemblyUnit.xLidsConveyorCmd
        OR (
            xPairSorterOutputPermit
            AND fbPairDiverter.xPusherZoneConveyorCmd
        )
    );

FIO.xAssemblyLidsPositionerRaiseCmd :=
    FALSE;

FIO.xAssemblyMoveXCmd :=
    xOutputPermit
    AND fbTwinCellOperatorControl.xRun
    AND fbAssemblyUnit.xMoveXCmd;

FIO.xAssemblyMoveZCmd :=
    xOutputPermit
    AND fbTwinCellOperatorControl.xRun
    AND fbAssemblyUnit.xMoveZCmd;

// =============================================================
// 11. SAFE FIO OUTPUT BOUNDARY — PART 2
// =============================================================

// Packout
FIO.xPackoutBufferConveyor1Cmd :=
    xOutputPermit
    AND fbPackoutLoader.xBufferConveyor1Cmd;

FIO.xPackoutBufferConveyor2Cmd :=
    xOutputPermit
    AND fbPackoutLoader.xBufferConveyor2Cmd;

FIO.xPackoutBufferConveyor3Cmd :=
    xOutputPermit
    AND fbPackoutLoader.xBufferConveyor3Cmd;
FIO.xPackoutCarrierConveyorCmd :=
    xOutputPermit
    AND fbPackoutCarrierStation.xCarrierConveyorCmd;

FIO.xPackoutCarrierEmitterCmd :=
    xOutputPermit
    AND fbPackoutCarrierStation.xCarrierEmitterCmd;

FIO.xPackoutCarrierInfeedConveyorCmd :=
    xOutputPermit
    AND fbPackoutCarrierStation.xCarrierInfeedConveyorCmd;
FIO.xPackoutGrabCmd :=
    xOutputPermit
    AND fbPackoutLoader.xGrabCmd;
FIO.xPackoutMoveXCmd :=
    xOutputPermit
    AND fbPackoutLoader.xMoveXCmd;
FIO.xPackoutMoveZCmd :=
    xOutputPermit
    AND fbPackoutLoader.xMoveZCmd;
FIO.xPackoutPickConveyorCmd :=
    xOutputPermit
    AND fbPackoutLoader.xPickConveyorCmd;

// Tank and transfer
IF xOutputPermit
    AND fbBatchStorageUnit.xTankDischargeValveCmd
THEN
    FIO.rTankDischargeValveCmdV := 10.0;
ELSE
    FIO.rTankDischargeValveCmdV := 0.0;
END_IF

IF xOutputPermit
    AND fbBatchStorageUnit.xTankFillValveCmd
THEN
    FIO.rTankFillValveCmdV := 10.0;
ELSE
    FIO.rTankFillValveCmdV := 0.0;
END_IF
FIO.xTankTransferConveyor1Cmd :=
    xOutputPermit
    AND fbBatchStorageUnit.xTankTransferConveyorsCmd;

FIO.xTankTransferConveyor2Cmd :=
    xOutputPermit
    AND fbBatchStorageUnit.xTankTransferConveyorsCmd;

FIO.xTankTransferConveyor3Cmd :=
    xOutputPermit
    AND fbBatchStorageUnit.xTankTransferConveyorsCmd;

FIO.xTankTransferConveyor4Cmd :=
    xOutputPermit
    AND fbBatchStorageUnit.xTankTransferConveyorsCmd;

// Permit for Storage and racking
xStorageOutputPermit :=
    FIO.xFactoryIORunning
    AND fbBatchStorageOperatorControl.xRun
    AND fbPlantCoordinator.xRunning
    AND NOT fbBatchStorageUnit.xStorageFaulted
    AND xOutputPermit;
	
// Storage and rack
// Storage and rack
IF xStorageOutputPermit THEN
    FIO.wStorageTargetPositionCmd :=
        fbBatchStorageUnit.wStorageTargetPositionCmd;
ELSE
    // Factory I/O target zero stops the numerical crane
    // at its current position.
    FIO.wStorageTargetPositionCmd := 0;
END_IF

FIO.xStorageEntryConveyorCmd :=
    xStorageOutputPermit
    AND fbBatchStorageUnit.xStorageEntryConveyorCmd;

FIO.xStorageExitConveyorCmd := FALSE;
FIO.xStorageExitRemoverCmd := FALSE;

FIO.xStorageForksLeftCmd :=
    xStorageOutputPermit
    AND fbBatchStorageUnit.xStorageForksLeftCmd;

FIO.xStorageForksRightCmd :=
    xStorageOutputPermit
    AND fbBatchStorageUnit.xStorageForksRightCmd;

FIO.xStorageLiftCmd :=
    xStorageOutputPermit
    AND fbBatchStorageUnit.xStorageLiftCmd;

FIO.xStorageLoadConveyorCmd :=
    xStorageOutputPermit
    AND fbBatchStorageUnit.xStorageLoadConveyorCmd;

FIO.xStorageUnloadConveyorCmd := FALSE;

// Packout stack light
FIO.xPackoutStackGreenCmd  := FIO.xMasterStackGreenCmd;
FIO.xPackoutStackRedCmd    := FIO.xMasterStackRedCmd;
FIO.xPackoutStackYellowCmd := FIO.xMasterStackYellowCmd;

// Plant stack light
FIO.xPlantStackGreenCmd  := FIO.xMasterStackGreenCmd;
FIO.xPlantStackRedCmd    := FIO.xMasterStackRedCmd;
FIO.xPlantStackYellowCmd := FIO.xMasterStackYellowCmd;

// Storage stack light
FIO.xStorageStackGreenCmd  := FIO.xMasterStackGreenCmd;
FIO.xStorageStackRedCmd    := FIO.xMasterStackRedCmd;
FIO.xStorageStackYellowCmd := FIO.xMasterStackYellowCmd;

// Tank stack light
FIO.xTankStackGreenCmd  := FIO.xMasterStackGreenCmd;
FIO.xTankStackRedCmd    := FIO.xMasterStackRedCmd;
FIO.xTankStackYellowCmd := FIO.xMasterStackYellowCmd;

END_PROGRAM

// Device/Application/POUs/FB_AssemblyUnit
FUNCTION_BLOCK FB_AssemblyUnit
VAR_INPUT
    xBaseAtPlace             : BOOL;
    xBaseClamped             : BOOL;
    xBasesPositionerAtLimit  : BOOL;
    xEnable                  : BOOL;
    xItemDetected            : BOOL;
    xLidAtPlace              : BOOL;
    xLidClamped              : BOOL;
    xMovingX                 : BOOL;
    xMovingZ                 : BOOL;
    xProductAtOutfeed        : BOOL;
    xProductTransferAck      : BOOL;
    xReset                   : BOOL;
    xRun                     : BOOL;
END_VAR

VAR_OUTPUT
    diProductCount              : DINT;
    eState                      : E_AssemblerState :=
        E_AssemblerState.Stopped;
    uiFaultCode                 : UINT;

    xBaseClampCmd               : BOOL;
    xBasesConveyorCmd           : BOOL;
    xBasesPositionerRaiseCmd    : BOOL;
    xBusy                       : BOOL;
    xFaulted                    : BOOL;
    xGrabCmd                    : BOOL;
    xLidClampCmd                : BOOL;
    xLidsConveyorCmd            : BOOL;
    xMoveXCmd                   : BOOL;
    xMoveZCmd                   : BOOL;
    xPairAck                    : BOOL;
    xPairReady                  : BOOL;
    xProductReq                 : BOOL;
    xReady                      : BOOL;
END_VAR

VAR
    fbAssemblerCell      : FB_AssemblerCell;
    xProductPending      : BOOL;
    xWaitForOutfeedClear : BOOL;
END_VAR

// =============================================================
// ASSEMBLER CELL
// =============================================================

fbAssemblerCell(
    tClampTimeout := T#5S,
    tFeedTimeout := T#10M,
    tGrabSettle := T#300MS,
    tHomeSettle := T#500MS,
    tMotionTimeout := T#10S,
    tProductExitTimeout := T#30S,
    tReleaseSettle := T#300MS,

    xBaseAtPlace := xBaseAtPlace,
    xBaseClamped := xBaseClamped,
    xBasesPositionerAtLimit := xBasesPositionerAtLimit,
    xEnable := xEnable AND xRun,
    xItemDetected := xItemDetected,
    xLidAtPlace := xLidAtPlace,
    xLidClamped := xLidClamped,
    xMovingX := xMovingX,
    xMovingZ := xMovingZ,
    xPartLeaving := xProductAtOutfeed,
    xReset := xReset
);

// =============================================================
// PHYSICAL COMMAND AND STATUS BOUNDARY
// =============================================================

diProductCount :=
    fbAssemblerCell.diProductsCompleted;

eState :=
    fbAssemblerCell.eState;

uiFaultCode :=
    fbAssemblerCell.uiFaultCode;

xBaseClampCmd :=
    fbAssemblerCell.xBaseClampCmd;

xBasesConveyorCmd :=
    fbAssemblerCell.xBasesConveyorCmd;

xBasesPositionerRaiseCmd :=
    fbAssemblerCell.xBasesPositionerRaiseCmd;

xFaulted :=
    fbAssemblerCell.xFaulted;

xGrabCmd :=
    fbAssemblerCell.xGrabCmd;

xLidClampCmd :=
    fbAssemblerCell.xLidClampCmd;

xLidsConveyorCmd :=
    fbAssemblerCell.xLidsConveyorCmd;

xMoveXCmd :=
    fbAssemblerCell.xMoveXCmd;

xMoveZCmd :=
    fbAssemblerCell.xMoveZCmd;

// =============================================================
// UNIT-TO-UNIT HANDSHAKES
// =============================================================

xPairAck := FALSE;
xPairReady := FALSE;
xProductReq := FALSE;
xReady := FALSE;

// Reset clears only the wrapper transaction memory.
// The child cell receives the same reset above.
IF xReset THEN
    xProductPending := FALSE;
    xWaitForOutfeedClear := FALSE;

// A complete disable abandons the pending transaction.
ELSIF NOT xEnable THEN
    xProductPending := FALSE;
    xWaitForOutfeedClear := FALSE;

ELSIF xRun THEN
    // Both physical arrival proofs acknowledge the P10-to-P11
    // pair transfer.
    xPairAck :=
        xBaseAtPlace
        AND xLidAtPlace;

    // Assembly can accept a new pair only while the proven cell
    // is waiting and both assembly positions are empty.
    xPairReady :=
        fbAssemblerCell.xReady
        AND NOT xBaseAtPlace
        AND NOT xLidAtPlace
        AND NOT xProductPending
        AND NOT xWaitForOutfeedClear;

    // Latch one completed product transaction at the outfeed.
    IF NOT xProductPending
        AND NOT xWaitForOutfeedClear
        AND xProductAtOutfeed
    THEN
        xProductPending := TRUE;
    END_IF;

    // Packout acknowledgement completes the transaction.
    IF xProductPending
        AND xProductTransferAck
    THEN
        xProductPending := FALSE;
        xWaitForOutfeedClear := TRUE;
    END_IF;

    // Require the outfeed proof to clear before accepting another
    // completed product.
    IF xWaitForOutfeedClear
        AND NOT xProductAtOutfeed
    THEN
        xWaitForOutfeedClear := FALSE;
    END_IF;

    xProductReq := xProductPending;
    xReady := xPairReady;
END_IF;

// Include both physical activity and the downstream transaction.
xBusy :=
    fbAssemblerCell.xBusy
    OR xProductPending
    OR xWaitForOutfeedClear;

// A fault removes every unit-boundary permission.
IF xFaulted THEN
    xPairAck := FALSE;
    xPairReady := FALSE;
    xProductReq := FALSE;
    xReady := FALSE;
END_IF;

END_FUNCTION_BLOCK

// Device/Application/POUs/FB_AssemblerCell
FUNCTION_BLOCK FB_AssemblerCell
VAR_INPUT
    tClampTimeout       : TIME;
    tFeedTimeout        : TIME;
    tGrabSettle         : TIME;
    tHomeSettle         : TIME;
    tMotionTimeout      : TIME;
    tProductExitTimeout : TIME;
    tReleaseSettle      : TIME;

    xBaseAtPlace            : BOOL;
    xBaseClamped            : BOOL;
    xBasesPositionerAtLimit : BOOL;
    xEnable                 : BOOL;
    xItemDetected           : BOOL;
    xLidAtPlace             : BOOL;
    xLidClamped             : BOOL;
    xMovingX                : BOOL;
    xMovingZ                : BOOL;
    xPartLeaving            : BOOL;
    xReset                  : BOOL;
END_VAR

VAR_OUTPUT
    diProductsCompleted : DINT;
    eState              : E_AssemblerState;
    uiFaultCode         : UINT;

    xBaseClampCmd            : BOOL;
    xBasesConveyorCmd        : BOOL;
    xBasesPositionerRaiseCmd : BOOL;
    xBusy                    : BOOL;
    xFaulted                 : BOOL;
    xGrabCmd                 : BOOL;
    xLidClampCmd             : BOOL;
    xLidsConveyorCmd         : BOOL;
    xMoveXCmd                : BOOL;
    xMoveZCmd                : BOOL;
    xProductCompletePulse    : BOOL;
    xReady                   : BOOL;
END_VAR

VAR
    ePreviousState : E_AssemblerState :=
        E_AssemblerState.Stopped;

    fbClampTimeout       : TON;
    fbFeedTimeout        : TON;
    fbGrabSettle         : TON;
    fbGrabTimeout        : TON;
    fbHomeSettle         : TON;
    fbMotionTimeout      : TON;
    fbProductExitTimeout : TON;
    fbReleaseSettle      : TON;

    rtPartLeaving : R_TRIG;

    xMotionObserved : BOOL;
    xStateChanged   : BOOL;
END_VAR

// =============================================================
// DEFAULT COMMANDS
//
// Every command must be deliberately enabled by the active state.
// =============================================================

xBaseClampCmd := FALSE;
xBasesConveyorCmd := FALSE;
xBasesPositionerRaiseCmd := FALSE;
xGrabCmd := FALSE;
xLidClampCmd := FALSE;
xLidsConveyorCmd := FALSE;
xMoveXCmd := FALSE;
xMoveZCmd := FALSE;
xProductCompletePulse := FALSE;

// =============================================================
// EDGE AND STATE-ENTRY DETECTION
// =============================================================

rtPartLeaving(CLK := xPartLeaving);

xStateChanged :=
    eState <> ePreviousState;

IF xStateChanged THEN
    ePreviousState := eState;
    xMotionObserved := FALSE;
END_IF;

// =============================================================
// STATE TIMERS
// =============================================================

fbClampTimeout(
    IN :=
        xEnable
        AND NOT xStateChanged
        AND (
            (eState = E_AssemblerState.ClampingParts)
            OR
            (eState = E_AssemblerState.ReleasingLidClamp)
        ),
    PT := tClampTimeout
);

fbFeedTimeout(
    IN :=
        xEnable
        AND NOT xStateChanged
        AND (eState = E_AssemblerState.WaitingForParts),
    PT := tFeedTimeout
);

fbGrabSettle(
    IN :=
        xEnable
        AND (eState = E_AssemblerState.GrippingLid)
        AND xItemDetected,
    PT := tGrabSettle
);

fbGrabTimeout(
    IN :=
        xEnable
        AND NOT xStateChanged
        AND (eState = E_AssemblerState.GrippingLid),
    PT := tMotionTimeout
);

fbHomeSettle(
    IN :=
        xEnable
        AND (eState = E_AssemblerState.Homing)
        AND NOT xMovingX
        AND NOT xMovingZ,
    PT := tHomeSettle
);

fbMotionTimeout(
    IN :=
        xEnable
        AND NOT xStateChanged
        AND (
            (eState = E_AssemblerState.Homing)
            OR
            (eState = E_AssemblerState.LoweringToLid)
            OR
            (eState = E_AssemblerState.LoweringToBase)
            OR
            (eState = E_AssemblerState.MovingToBase)
            OR
            (eState = E_AssemblerState.RaisingFromBase)
            OR
            (eState = E_AssemblerState.RaisingLid)
            OR
            (eState = E_AssemblerState.ReturningHome)
			OR
			(eState = E_AssemblerState.ReleasingProduct)
        ),
    PT := tMotionTimeout
);	

fbProductExitTimeout(
    IN :=
        xEnable
        AND NOT xStateChanged
        AND (eState = E_AssemblerState.WaitingForProductExit),
    PT := tProductExitTimeout
);

fbReleaseSettle(
    IN :=
        xEnable
        AND (eState = E_AssemblerState.ReleasingLid),
    PT := tReleaseSettle
);

// =============================================================
// RESET AND DISABLED CONDITIONS
// =============================================================

IF xReset THEN

    diProductsCompleted := 0;
    eState := E_AssemblerState.Stopped;
    uiFaultCode := 0;
    xMotionObserved := FALSE;

ELSIF NOT xEnable THEN

    // Fault state remains latched until Reset.
    IF eState <> E_AssemblerState.Faulted THEN
        eState := E_AssemblerState.Stopped;
    END_IF;

// =============================================================
// AUTOMATIC ASSEMBLY SEQUENCE
// =============================================================

ELSE

    CASE eState OF

        // -----------------------------------------------------
        // Begin every enabled run by returning the arm to its
        // default raised position above the lid.
        // -----------------------------------------------------

        E_AssemblerState.Stopped:

            eState := E_AssemblerState.Homing;

        // -----------------------------------------------------
        // Move X = FALSE: above the lid.
        // Move Z = FALSE: raised.
        //
        // The settle timer also handles the case where the arm
        // was already home and therefore produces no movement.
        // -----------------------------------------------------

        E_AssemblerState.Homing:

            IF fbHomeSettle.Q THEN
                eState := E_AssemblerState.WaitingForParts;

            ELSIF fbMotionTimeout.Q THEN
                uiFaultCode := 201;
                eState := E_AssemblerState.Faulted;
            END_IF;

        // -----------------------------------------------------
        // Keeps both positioners lowered while feeding material.
        // Each conveyor stops independently when its part
        // reaches the assembly position.
        // -----------------------------------------------------

		E_AssemblerState.WaitingForParts:
		
			// Keep both positioning assemblies lowered.
			// Feed each conveyor independently until its part arrives.
		
			xBasesConveyorCmd := NOT xBaseAtPlace;
			xLidsConveyorCmd := NOT xLidAtPlace;
		
			IF xBaseAtPlace
			AND xLidAtPlace THEN
		
				eState := E_AssemblerState.ClampingParts;
		
			ELSIF fbFeedTimeout.Q THEN
				uiFaultCode := 101;
				eState := E_AssemblerState.Faulted;
			END_IF;

        // -----------------------------------------------------
        // Secure both parts before the picker moves.
        // -----------------------------------------------------

        E_AssemblerState.ClampingParts:

			// Continue conveying each detected part into its clamp.
			// Stop each conveyor independently once clamped.
		
			xBaseClampCmd := TRUE;
			xBasesConveyorCmd := NOT xBaseClamped;
			xLidClampCmd := TRUE;
			xLidsConveyorCmd := NOT xLidClamped;
		
			IF xBaseClamped
			AND xLidClamped THEN
		
				eState := E_AssemblerState.LoweringToLid;
		
			ELSIF fbClampTimeout.Q THEN
				uiFaultCode := 102;
				eState := E_AssemblerState.Faulted;
			END_IF;

        // -----------------------------------------------------
        // Lower the picker onto the clamped lid.
        // -----------------------------------------------------

        E_AssemblerState.LoweringToLid:

            xBaseClampCmd := TRUE;
            
            xLidClampCmd := TRUE;
            
            xMoveZCmd := TRUE;

            IF xMovingZ THEN
                xMotionObserved := TRUE;
            END_IF;

            IF xMotionObserved AND NOT xMovingZ THEN
                eState := E_AssemblerState.GrippingLid;

            ELSIF fbMotionTimeout.Q THEN
                uiFaultCode := 202;
                eState := E_AssemblerState.Faulted;
            END_IF;

        // -----------------------------------------------------
        // Energise the suction cup and confirm the lid.
        // -----------------------------------------------------

        E_AssemblerState.GrippingLid:

            xBaseClampCmd := TRUE;
            
            xGrabCmd := TRUE;
            xLidClampCmd := TRUE;
            
            xMoveZCmd := TRUE;

            IF fbGrabSettle.Q THEN
                eState := E_AssemblerState.ReleasingLidClamp;

            ELSIF fbGrabTimeout.Q THEN
                uiFaultCode := 203;
                eState := E_AssemblerState.Faulted;
            END_IF;

        // -----------------------------------------------------
        // Release the lid clamp while suction retains the lid.
        // -----------------------------------------------------

        E_AssemblerState.ReleasingLidClamp:

            xBaseClampCmd := TRUE;
            
            xGrabCmd := TRUE;
            
            xMoveZCmd := TRUE;

            IF NOT xLidClamped THEN
                eState := E_AssemblerState.RaisingLid;

            ELSIF fbClampTimeout.Q THEN
                uiFaultCode := 204;
                eState := E_AssemblerState.Faulted;
            END_IF;

        // -----------------------------------------------------
        // Raise the collected lid.
        // -----------------------------------------------------

        E_AssemblerState.RaisingLid:

            xBaseClampCmd := TRUE;
            
            xGrabCmd := TRUE;
            

            IF xMovingZ THEN
                xMotionObserved := TRUE;
            END_IF;

            IF xMotionObserved AND NOT xMovingZ THEN
                eState := E_AssemblerState.MovingToBase;

            ELSIF fbMotionTimeout.Q THEN
                uiFaultCode := 205;
                eState := E_AssemblerState.Faulted;
            END_IF;

        // -----------------------------------------------------
        // Transfer from the home position above the lid to the
        // assembly position above the base.
        // -----------------------------------------------------

        E_AssemblerState.MovingToBase:

            xBaseClampCmd := TRUE;
            
            xGrabCmd := TRUE;
            
            xMoveXCmd := TRUE;

            IF xMovingX THEN
                xMotionObserved := TRUE;
            END_IF;

            IF xMotionObserved AND NOT xMovingX THEN
                eState := E_AssemblerState.LoweringToBase;

            ELSIF fbMotionTimeout.Q THEN
                uiFaultCode := 206;
                eState := E_AssemblerState.Faulted;
            END_IF;

        // -----------------------------------------------------
        // Lower the lid onto the clamped base.
        // -----------------------------------------------------

        E_AssemblerState.LoweringToBase:

            xBaseClampCmd := TRUE;
            
            xGrabCmd := TRUE;
            
            xMoveXCmd := TRUE;
            xMoveZCmd := TRUE;

            IF xMovingZ THEN
                xMotionObserved := TRUE;
            END_IF;

            IF xMotionObserved AND NOT xMovingZ THEN
                eState := E_AssemblerState.ReleasingLid;

            ELSIF fbMotionTimeout.Q THEN
                uiFaultCode := 207;
                eState := E_AssemblerState.Faulted;
            END_IF;

        // -----------------------------------------------------
        // Release suction. Correct physical alignment causes
        // Factory I/O to join the lid and base automatically.
        // -----------------------------------------------------

        E_AssemblerState.ReleasingLid:

            xBaseClampCmd := TRUE;
            
            
            xMoveXCmd := TRUE;
            xMoveZCmd := TRUE;

            IF fbReleaseSettle.Q THEN
                eState := E_AssemblerState.RaisingFromBase;
            END_IF;

        // -----------------------------------------------------
        // Raise clear of the assembled product.
        // -----------------------------------------------------

        E_AssemblerState.RaisingFromBase:

            xBaseClampCmd := TRUE;
            
            
            xMoveXCmd := TRUE;

            IF xMovingZ THEN
                xMotionObserved := TRUE;
            END_IF;

            IF xMotionObserved AND NOT xMovingZ THEN
                eState := E_AssemblerState.ReturningHome;

            ELSIF fbMotionTimeout.Q THEN
                uiFaultCode := 208;
                eState := E_AssemblerState.Faulted;
            END_IF;

        // -----------------------------------------------------
        // Return to the default position above the lid.
        // -----------------------------------------------------

        E_AssemblerState.ReturningHome:

            xBaseClampCmd := TRUE;
            
            

            IF xMovingX THEN
                xMotionObserved := TRUE;
            END_IF;

            IF xMotionObserved AND NOT xMovingX THEN
                eState := E_AssemblerState.ReleasingProduct;

            ELSIF fbMotionTimeout.Q THEN
                uiFaultCode := 209;
                eState := E_AssemblerState.Faulted;
            END_IF;

        // -----------------------------------------------------
        // Release the base clamp and raise the base positioner.
        // The finished product exits along the base conveyor.
        // -----------------------------------------------------

        E_AssemblerState.ReleasingProduct:

			// Release the base clamp through its default FALSE command
			// and raise the positioning assembly clear of the product.
		
			xBasesPositionerRaiseCmd := TRUE;
		
			IF xBasesPositionerAtLimit THEN
				eState := E_AssemblerState.WaitingForProductExit;
		
			ELSIF fbMotionTimeout.Q THEN
				uiFaultCode := 210; // Base positioner failed to raise.
				eState := E_AssemblerState.Faulted;
			END_IF;

        // -----------------------------------------------------
        // Wait for the downstream sensor. Its rising edge gives
        // exactly one count for each completed product.
        // -----------------------------------------------------

        E_AssemblerState.WaitingForProductExit:

			// Once clearance has been confirmed, keep the conveyors
			// running without continuously depending on the limit signal.
		
			xBasesConveyorCmd := TRUE;
			xBasesPositionerRaiseCmd := TRUE;
			xLidsConveyorCmd := NOT xLidAtPlace;
		
			IF rtPartLeaving.Q THEN
		
				diProductsCompleted :=
					diProductsCompleted + 1;
		
				xProductCompletePulse := TRUE;
				eState := E_AssemblerState.WaitingForParts;
		
			ELSIF fbMotionTimeout.Q THEN
				uiFaultCode := 301;
				eState := E_AssemblerState.Faulted;
			END_IF;

        // -----------------------------------------------------
        // Latched safe state.
        // -----------------------------------------------------

        E_AssemblerState.Faulted:

        // -----------------------------------------------------
        // Corrupted or unexpected enumeration value.
        // -----------------------------------------------------

        ELSE

            uiFaultCode := 999;
            eState := E_AssemblerState.Faulted;

    END_CASE;

END_IF;

// =============================================================
// STATUS OUTPUTS
// =============================================================

xFaulted :=
    eState = E_AssemblerState.Faulted;

xReady :=
    xEnable
    AND (eState = E_AssemblerState.WaitingForParts);

xBusy :=
    xEnable
    AND (eState <> E_AssemblerState.Stopped)
    AND (eState <> E_AssemblerState.WaitingForParts)
    AND (eState <> E_AssemblerState.Faulted);

// Ensure every physical command is de-energised after a fault.
IF xFaulted THEN
    xBaseClampCmd := FALSE;
    xBasesConveyorCmd := FALSE;
    xBasesPositionerRaiseCmd := FALSE;
    xGrabCmd := FALSE;
    xLidClampCmd := FALSE;
    xLidsConveyorCmd := FALSE;
    xMoveXCmd := FALSE;
    xMoveZCmd := FALSE;
END_IF;

END_FUNCTION_BLOCK

// Device/Application/POUs/FB_UnitOperatorControl
FUNCTION_BLOCK FB_UnitOperatorControl
VAR_INPUT
    xEmergencyStopHealthy   : BOOL;
    xLocalModeSelected      : BOOL;
    xLocalResetPB           : BOOL;
    xLocalStartPB           : BOOL;
    xLocalStopHealthy       : BOOL;
	xMasterAutoModeActive   : BOOL;
    xMasterEnable           : BOOL;
	xMasterManualModeActive : BOOL;
    xMasterModeSelected     : BOOL;
    xMasterResetPulse       : BOOL;
    xMasterRun              : BOOL;
    xTransferActive         : BOOL;
END_VAR
VAR_OUTPUT
    xEnable           : BOOL;
    xLocalModeActive  : BOOL;
    xMasterModeActive : BOOL;
    xResetPulse       : BOOL;
    xRun              : BOOL;
END_VAR
VAR
    fbLocalResetEdge : R_TRIG;
    fbLocalStartEdge : R_TRIG;
    fbMasterRunEdge  : R_TRIG;
    xModeValid       : BOOL;
    xRunLatched      : BOOL;
END_VAR

fbLocalResetEdge(CLK := xLocalResetPB);
fbLocalStartEdge(CLK := xLocalStartPB);
fbMasterRunEdge(CLK := xMasterRun);

// Exactly one unit-panel operating mode must be selected.
xModeValid :=
    xLocalModeSelected XOR xMasterModeSelected;

xLocalModeActive :=
    xLocalModeSelected
    AND NOT xMasterModeSelected;

xMasterModeActive :=
    xMasterModeSelected
    AND NOT xLocalModeSelected;

// One-scan default.
xResetPulse := FALSE;

// Any immediate interlock loss cancels the run latch.
IF NOT xEmergencyStopHealthy
    OR NOT xLocalStopHealthy
    OR NOT xMasterEnable
    OR NOT xModeValid
THEN
    xRunLatched := FALSE;

// Local Reset and Start are accepted in Local mode.
ELSIF xLocalModeActive THEN
    IF fbLocalResetEdge.Q AND NOT xTransferActive THEN
        xResetPulse := TRUE;
        xRunLatched := FALSE;

    ELSIF fbLocalStartEdge.Q THEN
        xRunLatched := TRUE;
    END_IF

// MASTER Start initially starts the zone.
// Following a local Stop, the local Start button deliberately
// allows only this zone to rejoin the running plant.
ELSIF xMasterModeActive THEN
    xResetPulse := xMasterResetPulse;

    IF NOT xMasterRun THEN
        xRunLatched := FALSE;

    ELSIF fbMasterRunEdge.Q THEN
        xRunLatched := TRUE;

    ELSIF fbLocalStartEdge.Q THEN
        xRunLatched := TRUE;
    END_IF
END_IF

// Both the MASTER selector and the unit selector must agree.
xEnable :=
    xEmergencyStopHealthy
    AND xLocalStopHealthy
    AND xMasterEnable
    AND xModeValid
    AND (
        (xLocalModeActive AND xMasterManualModeActive)
        OR
        (xMasterModeActive AND xMasterAutoModeActive)
    );

// Select the permitted run authority.
IF xLocalModeActive THEN
    xRun := xEnable AND xRunLatched;

ELSIF xMasterModeActive THEN
    xRun :=
        xEnable
        AND xMasterRun
        AND xRunLatched;

ELSE
    xRun := FALSE;
END_IF

END_FUNCTION_BLOCK

// Device/Application/POUs/FB_BatchStorageUnit
FUNCTION_BLOCK FB_BatchStorageUnit
VAR_INPUT
    rTankLevelV             : REAL;
	wStorageHomePosition    : WORD := 55;
    xStorageCraneAtHome     : BOOL;
    xStorageForkAtLeft      : BOOL;
    xStorageForkAtMiddle    : BOOL;
    xStorageForkAtRight     : BOOL;
    xStorageMovingX         : BOOL;
    xStorageMovingZ         : BOOL;
    xStorageProductAtLoad   : BOOL;
    xEnable                 : BOOL;
    xPackoutPalletAtLoad    : BOOL;
    xPackoutProductLoaded   : BOOL;
    xProductTransferReq     : BOOL;
    xReset                  : BOOL;
    xRun                    : BOOL;
    xStorageAtEntry         : BOOL;
    xTankCarrierAtFill      : BOOL;
    xTankLevelHighHigh      : BOOL;
END_VAR

VAR_OUTPUT
    eState                    : E_BatchStorageState :=
                                    E_BatchStorageState.Stopped;
	eStorageState             : E_StorageState :=
                                        E_StorageState.Stopped;
    eTankState                : E_TankState :=
                                    E_TankState.Stopped;
    uiFaultCode               : UINT;
    uiRackFreeCount           : UINT;
    uiRackOccupiedCount       : UINT;
    uiRackReservedCount       : UINT;
    uiRackUnknownCount        : UINT;
	uiStorageFaultCode        : UINT;
    wRackReservedPosition     : WORD;
	wStorageTargetPositionCmd : WORD := 55;
    xBusy                     : BOOL;
    xFaulted                  : BOOL;
    xProductTransferAck       : BOOL;
    xProductTransferReady     : BOOL;
    xRackCommitAck            : BOOL;
    xRackFull                 : BOOL;
    xRackReservationValid     : BOOL;
    xReady                    : BOOL;
	xStorageBusy 			  : BOOL;
	xStorageDepositComplete   : BOOL;
	xStorageEntryConveyorCmd  : BOOL; 
	xStorageFaulted           : BOOL; 
	xStorageForksLeftCmd      : BOOL;
	xStorageForksRightCmd     : BOOL;
	xStorageLiftCmd           : BOOL; 
	xStorageLoadConveyorCmd   : BOOL;
	xStorageReady             : BOOL;
    xStorageStoreComplete     : BOOL;
    xTankDischargeValveCmd    : BOOL;
    xTankFillValveCmd         : BOOL;
    xTankTransferConveyorsCmd : BOOL;
END_VAR

VAR
    fbRackManager      : FB_RackManager;
	fbStorage          : FB_Storage;
    fbTank             : FB_Tank;
    xCarrierAccepted   : BOOL;
    xTransactionActive : BOOL;
END_VAR

// Tank batch production and discharge.
fbTank(
    rEmptySetpointPct := 5.0,
    rFillSetpointPct := 80.0,
    rLevelPct := rTankLevelV * 10.0,
    tDischargeTimeout := T#30M,
	tFillTimeout := T#30M,

    xDischargePermit :=
        xRun
        AND
        (eState = E_BatchStorageState.DischargingBatch),

    xEnable := xEnable,
    xLevelHighHigh := xTankLevelHighHigh,
    xReset := xReset,

    xStartBatchReq :=
        xRun
        AND (
            (eState = E_BatchStorageState.ReservingSlot)
            OR
            (eState = E_BatchStorageState.WaitingForBatch)
            OR
            (eState = E_BatchStorageState.DischargingBatch)
        )
);

eTankState := fbTank.eState;
xTankDischargeValveCmd := fbTank.xDischargeValveCmd;
xTankFillValveCmd := fbTank.xFillValveCmd;

// Rack inventory and reservation ownership.
fbRackManager(
    xCommitRequest :=
        eState = E_BatchStorageState.CommittingInventory,

    xEnable :=
        xEnable
        AND xRun,

    // Until the crane sequence provides a more precise deposit proof,
    // any reset after entering storage is handled conservatively.
    xReservationMayBeOccupied :=
        (eState = E_BatchStorageState.StoringProduct)
        OR
        (eState = E_BatchStorageState.CommittingInventory)
        OR
        (eState = E_BatchStorageState.WaitingForStorageComplete),

    xReserveRequest :=
        eState = E_BatchStorageState.ReservingSlot,

    xReset := xReset
);

// Automated rack-storage sequence.
fbStorage(
    tLiftTime := T#2S,
    tLowerTime := T#2S,
    tStepTimeout := T#2M,
    wHomePosition := wStorageHomePosition,
    wReservedPosition := fbRackManager.wReservedPosition,
    xCraneAtHome := xStorageCraneAtHome,
    xEnable := xEnable,
    xForkAtLeft := xStorageForkAtLeft,
    xForkAtMiddle := xStorageForkAtMiddle,
    xForkAtRight := xStorageForkAtRight,
    xMovingX := xStorageMovingX,
    xMovingZ := xStorageMovingZ,
    xProductAtLoad := xStorageProductAtLoad,
    xReservationValid := fbRackManager.xReservationValid,
    xReset := xReset,
    xRun := xRun,
    xStoreRequest :=
        eState = E_BatchStorageState.StoringProduct
);

// Publish storage status and requested commands.
eStorageState := fbStorage.eState;
uiStorageFaultCode := fbStorage.uiFaultCode;
wStorageTargetPositionCmd := fbStorage.wTargetPositionCmd;
xStorageBusy := fbStorage.xBusy;
xStorageDepositComplete := fbStorage.xDepositComplete;
xStorageEntryConveyorCmd := fbStorage.xEntryConveyorCmd;
xStorageFaulted := fbStorage.xFaulted;
xStorageForksLeftCmd := fbStorage.xForksLeftCmd;
xStorageForksRightCmd := fbStorage.xForksRightCmd;
xStorageLiftCmd := fbStorage.xLiftCmd;
xStorageLoadConveyorCmd := fbStorage.xLoadConveyorCmd;
xStorageReady := fbStorage.xReady;
xStorageStoreComplete := fbStorage.xStoreComplete;

// Publish the rack manager's authoritative values.
uiRackFreeCount := fbRackManager.uiFreeCount;
uiRackOccupiedCount := fbRackManager.uiOccupiedCount;
uiRackReservedCount := fbRackManager.uiReservedCount;
uiRackUnknownCount := fbRackManager.uiUnknownCount;
wRackReservedPosition := fbRackManager.wReservedPosition;
xRackCommitAck := fbRackManager.xCommitAck;
xRackFull := fbRackManager.xRackFull;
xRackReservationValid := fbRackManager.xReservationValid;

// Safe output defaults.
xTankTransferConveyorsCmd := FALSE;

IF xReset THEN
    eState := E_BatchStorageState.Stopped;
    uiFaultCode := 0;
    xBusy := FALSE;
    xCarrierAccepted := FALSE;
    xFaulted := FALSE;
    xProductTransferAck := FALSE;
    xProductTransferReady := FALSE;
    xReady := FALSE;
    xTransactionActive := FALSE;

ELSIF NOT xEnable THEN
    // Preserve the transaction and reservation while the zone is stopped.
    xBusy :=
        xTransactionActive
        OR (eState = E_BatchStorageState.DischargingBatch)
        OR (eState = E_BatchStorageState.StoringProduct)
        OR (eState = E_BatchStorageState.CommittingInventory);

    xFaulted := eState = E_BatchStorageState.Faulted;
    xProductTransferAck := xCarrierAccepted;
    xProductTransferReady := FALSE;
    xReady := FALSE;

ELSE
    CASE eState OF

        E_BatchStorageState.Stopped:
            xBusy := FALSE;
            xFaulted := FALSE;
            xProductTransferAck := FALSE;
            xProductTransferReady := FALSE;
            xReady := FALSE;

            eState := E_BatchStorageState.ReservingSlot;


        E_BatchStorageState.ReservingSlot:
			xBusy := FALSE;
			xProductTransferAck := FALSE;
			xProductTransferReady := FALSE;
			xReady := FALSE;
		
			IF fbRackManager.xReserveAck THEN
				IF fbRackManager.xReservationValid THEN
					xReady := TRUE;
					eState := E_BatchStorageState.WaitingForBatch;
		
				ELSIF fbRackManager.xRackFull THEN
					uiFaultCode := 620;
					xFaulted := TRUE;
					eState := E_BatchStorageState.Faulted;
				END_IF;
			END_IF


        E_BatchStorageState.WaitingForBatch:
            xBusy := xTransactionActive;
            xReady := TRUE;

            // P9 accepts only one loaded carrier at a time.
            xProductTransferReady :=
				fbTank.xBatchReady
				AND xRun
				AND NOT xTransactionActive
				AND NOT xTankCarrierAtFill;

            IF xProductTransferReq
                AND xProductTransferReady
                AND xPackoutPalletAtLoad
                AND xPackoutProductLoaded
            THEN
                xTransactionActive := TRUE;
                xBusy := TRUE;
            END_IF
			
			// Move the accepted loaded carrier from Packout to the tank.
			xTankTransferConveyorsCmd :=
				xRun
				AND xTransactionActive
				AND NOT xTankCarrierAtFill;

            // Physical arrival at the tank station acknowledges transfer.
            IF xRun
				AND xTransactionActive
				AND xTankCarrierAtFill
			THEN
				xCarrierAccepted := TRUE;
				xProductTransferAck := TRUE;
			END_IF

            // Hold acknowledgement until the upstream request clears.
            IF xRun
				AND xCarrierAccepted
				AND NOT xProductTransferReq
			THEN
				xProductTransferAck := FALSE;
				xCarrierAccepted := FALSE;
				eState := E_BatchStorageState.DischargingBatch;
			END_IF


        E_BatchStorageState.DischargingBatch:
            xBusy := TRUE;
            xProductTransferReady := FALSE;
            xReady := FALSE;

            // Temporary proof that the tank has received material.
            // Real filling/discharge thresholds will come from FB_Tank.
            IF xRun AND fbTank.xDischargeComplete THEN
				eState := E_BatchStorageState.StoringProduct;
			END_IF


        E_BatchStorageState.StoringProduct:
            xBusy := TRUE;
            xProductTransferReady := FALSE;
            xReady := FALSE;

           // Move the discharged carrier from the tank to the
			// single storage-entry staging position.
			xTankTransferConveyorsCmd :=
				xRun
				AND NOT xStorageAtEntry;
			
			// Inventory is committed only after the storage module
            // has deposited the carrier and returned home.
            IF xRun AND fbStorage.xStoreComplete THEN
                eState :=
                    E_BatchStorageState.CommittingInventory;
            END_IF


        E_BatchStorageState.CommittingInventory:
			xBusy := TRUE;
			xProductTransferReady := FALSE;
			xReady := FALSE;
		
			IF xRun AND fbRackManager.xCommitAck THEN
				eState :=
					E_BatchStorageState.WaitingForStorageComplete;
			END_IF

        E_BatchStorageState.WaitingForStorageComplete:
			xBusy := FALSE;
			xProductTransferReady := FALSE;
			xReady := FALSE;
		
			IF xRun THEN
				// Begin reservation for the next single plant transaction.
				xTransactionActive := FALSE;
				eState := E_BatchStorageState.ReservingSlot;
			END_IF


        E_BatchStorageState.Faulted:
            xBusy := FALSE;
            xFaulted := TRUE;
            xProductTransferAck := FALSE;
            xProductTransferReady := FALSE;
            xReady := FALSE;


    ELSE
        uiFaultCode := 699;
        xFaulted := TRUE;
        eState := E_BatchStorageState.Faulted;

    END_CASE
END_IF

IF fbRackManager.xFaulted THEN
    uiFaultCode := 621;
    xFaulted := TRUE;
    eState := E_BatchStorageState.Faulted;
END_IF;

IF fbTank.xFaulted THEN
    uiFaultCode := 610;
    xFaulted := TRUE;
    eState := E_BatchStorageState.Faulted;
END_IF

IF fbStorage.xFaulted THEN
    uiFaultCode := 630;
    xFaulted := TRUE;
    eState := E_BatchStorageState.Faulted;
END_IF

IF xFaulted THEN
    xBusy := FALSE;
    xProductTransferAck := FALSE;
    xProductTransferReady := FALSE;
    xReady := FALSE;
END_IF

END_FUNCTION_BLOCK

// Device/Application/POUs/FB_Tank
FUNCTION_BLOCK FB_Tank
VAR_INPUT
    rEmptySetpointPct : REAL := 5.0;
    rFillSetpointPct  : REAL := 80.0;
    rLevelPct         : REAL;

    tDischargeTimeout : TIME := T#2M;
    tFillTimeout      : TIME := T#2M;

    xDischargePermit  : BOOL;
    xEnable           : BOOL;
    xLevelHighHigh    : BOOL;
    xReset            : BOOL;
    xStartBatchReq    : BOOL;
END_VAR

VAR_OUTPUT
    eState                   : E_TankState :=
        E_TankState.Stopped;

    xBatchReady              : BOOL;
    xDischargeComplete       : BOOL;
    xDischargeTimeoutFault   : BOOL;
    xDischargeValveCmd       : BOOL;
    xFaulted                 : BOOL;
    xFillTimeoutFault        : BOOL;
    xFillValveCmd            : BOOL;
    xHighHighFault           : BOOL;
    xReady                   : BOOL;
END_VAR

VAR
    fbDischargeTimeout : TON;
    fbFillTimeout      : TON;
END_VAR

// Timeouts only run while their corresponding operation is active.
fbDischargeTimeout(
    IN :=
        xEnable
        AND NOT xReset
        AND (eState = E_TankState.Discharging),
    PT := tDischargeTimeout
);

fbFillTimeout(
    IN :=
        xEnable
        AND NOT xReset
        AND (eState = E_TankState.Filling),
    PT := tFillTimeout
);

// Safe one-scan defaults.
xBatchReady := FALSE;
xDischargeComplete := FALSE;
xDischargeValveCmd := FALSE;
xFillValveCmd := FALSE;
xReady := FALSE;

IF xReset THEN
    eState := E_TankState.Stopped;

    xDischargeTimeoutFault := FALSE;
    xFillTimeoutFault := FALSE;
    xHighHighFault := xLevelHighHigh;

ELSE
    // High-high is latched until a healthy reset.
    IF xLevelHighHigh THEN
        xHighHighFault := TRUE;
    END_IF

    IF fbDischargeTimeout.Q THEN
        xDischargeTimeoutFault := TRUE;
    END_IF

    IF fbFillTimeout.Q THEN
        xFillTimeoutFault := TRUE;
    END_IF

    xFaulted :=
        xDischargeTimeoutFault
        OR xFillTimeoutFault
        OR xHighHighFault;

    IF xFaulted THEN
        eState := E_TankState.Faulted;

    ELSIF xEnable THEN
        CASE eState OF

            E_TankState.Stopped:
                IF rLevelPct >= rFillSetpointPct THEN
                    eState := E_TankState.BatchReady;
                ELSE
                    eState := E_TankState.Idle;
                END_IF


            E_TankState.Idle:
                IF xStartBatchReq THEN
                    eState := E_TankState.Filling;
                END_IF


            E_TankState.Filling:
                IF rLevelPct >= rFillSetpointPct THEN
                    eState := E_TankState.BatchReady;
                ELSE
                    xFillValveCmd := TRUE;
                END_IF


            E_TankState.BatchReady:
                IF xDischargePermit THEN
                    eState := E_TankState.Discharging;
                END_IF


            E_TankState.Discharging:
                IF rLevelPct <= rEmptySetpointPct THEN
                    // Hold completion until the owner removes
                    // its discharge permit.
                    xDischargeComplete := TRUE;

                    IF NOT xDischargePermit THEN
                        eState := E_TankState.Idle;
                    END_IF

                ELSIF xDischargePermit THEN
                    xDischargeValveCmd := TRUE;
                END_IF


            E_TankState.Faulted:
                // Reset is required to leave this state.


        ELSE
            xHighHighFault := TRUE;
            eState := E_TankState.Faulted;

        END_CASE
    END_IF
END_IF

// Publish persistent status after all state processing.
xFaulted :=
    xDischargeTimeoutFault
    OR xFillTimeoutFault
    OR xHighHighFault;

IF xFaulted THEN
    eState := E_TankState.Faulted;
    xDischargeComplete := FALSE;
    xDischargeValveCmd := FALSE;
    xFillValveCmd := FALSE;
END_IF

xBatchReady :=
    xEnable
    AND NOT xFaulted
    AND (eState = E_TankState.BatchReady);

xReady :=
    xEnable
    AND NOT xFaulted
    AND (eState = E_TankState.Idle);

END_FUNCTION_BLOCK

// Device/Application/POUs/FB_RackManager
FUNCTION_BLOCK FB_RackManager
VAR_INPUT
    xCommitRequest            : BOOL;
    xEnable                   : BOOL;
    xReservationMayBeOccupied : BOOL;
    xReserveRequest           : BOOL;
    xReset                    : BOOL;
END_VAR

VAR_OUTPUT
    aSlotState       : ARRAY[1..54] OF E_RackSlotState;
    uiFreeCount      : UINT;
    uiOccupiedCount  : UINT;
    uiReservedCount  : UINT;
    uiUnknownCount   : UINT;
    wReservedPosition : WORD;
    xCommitAck       : BOOL;
    xFaulted         : BOOL;
    xRackFull        : BOOL;
    xReservationValid : BOOL;
    xReserveAck      : BOOL;
END_VAR

VAR
    iSlot                 : INT;
    wCandidatePosition    : WORD;
    xInvalidOperationFault : BOOL;
END_VAR

// Acknowledgements remain active until their requests return low.
IF NOT xCommitRequest THEN
    xCommitAck := FALSE;
END_IF;

IF NOT xReserveRequest THEN
    xReserveAck := FALSE;
END_IF;

// Reset clears control faults without deleting occupied inventory.
IF xReset
    AND NOT xCommitRequest
    AND NOT xReserveRequest
THEN
    xInvalidOperationFault := FALSE;

    IF xReservationValid THEN
        IF (wReservedPosition >= 1)
            AND (wReservedPosition <= 54)
            AND (
                aSlotState[WORD_TO_INT(wReservedPosition)]
                = E_RackSlotState.Reserved
            )
        THEN
            // If material may already have been deposited, quarantine
            // the slot instead of incorrectly marking it free.
            IF xReservationMayBeOccupied THEN
                aSlotState[WORD_TO_INT(wReservedPosition)] :=
                    E_RackSlotState.Unknown;
            ELSE
                aSlotState[WORD_TO_INT(wReservedPosition)] :=
                    E_RackSlotState.Free;
            END_IF;

            wReservedPosition := 0;
            xReservationValid := FALSE;
        ELSE
            xInvalidOperationFault := TRUE;
        END_IF;
    END_IF;
END_IF;

// Reserve and commit must never be requested simultaneously.
IF xCommitRequest AND xReserveRequest THEN
    xInvalidOperationFault := TRUE;
END_IF;

xFaulted := xInvalidOperationFault;

IF xEnable AND NOT xFaulted THEN
    // Commit the current reservation only after physical deposit.
    IF xCommitRequest AND NOT xCommitAck THEN
        IF xReservationValid
            AND (wReservedPosition >= 1)
            AND (wReservedPosition <= 54)
            AND (
                aSlotState[WORD_TO_INT(wReservedPosition)]
                = E_RackSlotState.Reserved
            )
        THEN
            aSlotState[WORD_TO_INT(wReservedPosition)] :=
                E_RackSlotState.Occupied;

            wReservedPosition := 0;
            xCommitAck := TRUE;
            xReservationValid := FALSE;
        ELSE
            xInvalidOperationFault := TRUE;
        END_IF;

    // Select the first available rack position.
    ELSIF xReserveRequest AND NOT xReserveAck THEN
        IF xReservationValid THEN
            xInvalidOperationFault := TRUE;
        ELSE
            wCandidatePosition := 0;
            wReservedPosition := 0;

            FOR iSlot := 1 TO 54 DO
                IF (wCandidatePosition = 0)
                    AND (
                        aSlotState[iSlot]
                        = E_RackSlotState.Free
                    )
                THEN
                    wCandidatePosition := INT_TO_WORD(iSlot);
                END_IF;
            END_FOR;

            IF wCandidatePosition <> 0 THEN
                aSlotState[WORD_TO_INT(wCandidatePosition)] :=
                    E_RackSlotState.Reserved;

                wReservedPosition := wCandidatePosition;
                xReservationValid := TRUE;
            END_IF;

            // Acknowledge even when full; ReservationValid reports
            // whether a position was successfully obtained.
            xReserveAck := TRUE;
        END_IF;
    END_IF;
END_IF;

// Recalculate rack inventory every scan.
uiFreeCount := 0;
uiOccupiedCount := 0;
uiReservedCount := 0;
uiUnknownCount := 0;

FOR iSlot := 1 TO 54 DO
    CASE aSlotState[iSlot] OF
        E_RackSlotState.Free:
            uiFreeCount := uiFreeCount + 1;

        E_RackSlotState.Occupied:
            uiOccupiedCount := uiOccupiedCount + 1;

        E_RackSlotState.Reserved:
            uiReservedCount := uiReservedCount + 1;

        E_RackSlotState.Unknown:
            uiUnknownCount := uiUnknownCount + 1;
    END_CASE;
END_FOR;

xFaulted := xInvalidOperationFault;
xRackFull := uiFreeCount = 0;

END_FUNCTION_BLOCK

// Device/Application/POUs/FB_Storage
FUNCTION_BLOCK FB_Storage
VAR_INPUT
    tLiftTime         : TIME := T#2S;
    tLowerTime        : TIME := T#2S;
    tStepTimeout      : TIME := T#30S;
    wHomePosition     : WORD := 55;
    wReservedPosition : WORD;
    xCraneAtHome      : BOOL;
    xEnable           : BOOL;
    xForkAtLeft       : BOOL;
    xForkAtMiddle     : BOOL;
    xForkAtRight      : BOOL;
    xMovingX          : BOOL;
    xMovingZ          : BOOL;
    xProductAtLoad    : BOOL;
    xReservationValid : BOOL;
    xReset            : BOOL;
    xRun              : BOOL;
    xStoreRequest     : BOOL;
END_VAR

VAR_OUTPUT
    eState                 : E_StorageState :=
                                 E_StorageState.Stopped;
    uiFaultCode            : UINT;
    wTargetPositionCmd     : WORD := 55;
    xBusy                  : BOOL;
    xDepositComplete       : BOOL;
    xEntryConveyorCmd      : BOOL;
    xFaulted               : BOOL;
    xForksLeftCmd          : BOOL;
    xForksRightCmd         : BOOL;
    xLiftCmd               : BOOL;
    xLoadConveyorCmd       : BOOL;
    xReady                 : BOOL;
    xStepTimeoutFault      : BOOL;
    xStoreComplete         : BOOL;
END_VAR

VAR
    ePreviousState    : E_StorageState :=
                            E_StorageState.Stopped;
    fbLiftTimer       : TON;
    fbLowerTimer      : TON;
    fbStepTimeout     : TON;
    wActivePosition   : WORD;
    xCommandArmed     : BOOL;
    xMotionStarted    : BOOL;
    xReservationFault : BOOL;
    xStateChanged     : BOOL;
    xTimedStep        : BOOL;
END_VAR

// Vertical movements do not provide dedicated raised/lowered
// feedback, so their travel is deliberately timed.
fbLiftTimer(
    IN :=
        xEnable
        AND xRun
        AND (eState = E_StorageState.LiftingProduct),
    PT := tLiftTime
);

fbLowerTimer(
    IN :=
        xEnable
        AND xRun
        AND (eState = E_StorageState.LoweringProduct),
    PT := tLowerTime
);

// Safe Boolean defaults.
xEntryConveyorCmd := FALSE;
xForksLeftCmd := FALSE;
xForksRightCmd := FALSE;
xLiftCmd := FALSE;
xLoadConveyorCmd := FALSE;
xReady := FALSE;

// Reset returns the module to a known, non-moving baseline.
IF xReset THEN
    eState := E_StorageState.Stopped;
    uiFaultCode := 0;
    wActivePosition := 0;
    wTargetPositionCmd := wHomePosition;
    xCommandArmed := FALSE;
    xDepositComplete := FALSE;
    xMotionStarted := FALSE;
    xReservationFault := FALSE;
    xStepTimeoutFault := FALSE;
END_IF;

// A Store request must return low before another is accepted.
IF xReset OR xFaulted THEN
    xCommandArmed := FALSE;

ELSIF NOT xStoreRequest THEN
    xCommandArmed := TRUE;
END_IF;

xFaulted :=
    xReservationFault
    OR xStepTimeoutFault;

IF xFaulted THEN
    eState := E_StorageState.Faulted;
END_IF;

// Removing Run pauses the current state and removes all Boolean
// motion commands. The transaction itself remains preserved.
IF xEnable
    AND xRun
    AND NOT xReset
    AND NOT xFaulted
THEN
    CASE eState OF

        E_StorageState.Stopped:
            wTargetPositionCmd := wHomePosition;

            IF xCraneAtHome AND xForkAtMiddle THEN
                eState := E_StorageState.Idle;
            ELSE
                xMotionStarted := FALSE;
                eState := E_StorageState.ReturningHome;
            END_IF;


        E_StorageState.Idle:
            wTargetPositionCmd := wHomePosition;

            IF xStoreRequest AND xCommandArmed THEN
                IF xReservationValid
                    AND (wReservedPosition >= 1)
                    AND (wReservedPosition <= 54)
                THEN
                    wActivePosition := wReservedPosition;
                    xCommandArmed := FALSE;
                    xDepositComplete := FALSE;
                    eState := E_StorageState.ReceivingProduct;
                ELSE
                    uiFaultCode := 710;
                    xReservationFault := TRUE;
                END_IF;
            END_IF;


        E_StorageState.ReceivingProduct:
            IF xProductAtLoad THEN
                eState := E_StorageState.ExtendingToLoad;
            ELSE
                xEntryConveyorCmd := TRUE;
                xLoadConveyorCmd := TRUE;
            END_IF;


        E_StorageState.ExtendingToLoad:
            xForksLeftCmd := TRUE;

            IF xForkAtLeft THEN
                eState := E_StorageState.LiftingProduct;
            END_IF;


        E_StorageState.LiftingProduct:
            xForksLeftCmd := TRUE;
            xLiftCmd := TRUE;

            IF fbLiftTimer.Q THEN
                eState := E_StorageState.RetractingWithProduct;
            END_IF;


        E_StorageState.RetractingWithProduct:
            xLiftCmd := TRUE;

            IF xForkAtMiddle THEN
                xMotionStarted := FALSE;
                eState := E_StorageState.MovingToRack;
            END_IF;


        E_StorageState.MovingToRack:
            wTargetPositionCmd := wActivePosition;
            xLiftCmd := TRUE;

            IF xMovingX OR xMovingZ THEN
                xMotionStarted := TRUE;
            END_IF;

            IF xMotionStarted
                AND NOT xMovingX
                AND NOT xMovingZ
            THEN
                xMotionStarted := FALSE;
                eState := E_StorageState.ExtendingToRack;
            END_IF;


        E_StorageState.ExtendingToRack:
            wTargetPositionCmd := wActivePosition;
            xForksRightCmd := TRUE;
            xLiftCmd := TRUE;

            IF xForkAtRight THEN
                eState := E_StorageState.LoweringProduct;
            END_IF;


        E_StorageState.LoweringProduct:
            wTargetPositionCmd := wActivePosition;
            xForksRightCmd := TRUE;

            IF fbLowerTimer.Q THEN
                eState :=
                    E_StorageState.RetractingAfterDeposit;
            END_IF;


        E_StorageState.RetractingAfterDeposit:
            wTargetPositionCmd := wActivePosition;

            IF xForkAtMiddle THEN
                xDepositComplete := TRUE;
                xMotionStarted := FALSE;
                eState := E_StorageState.ReturningHome;
            END_IF;


        E_StorageState.ReturningHome:
            wTargetPositionCmd := wHomePosition;

            IF xMovingX OR xMovingZ THEN
                xMotionStarted := TRUE;
            END_IF;

            IF xForkAtMiddle
                AND (
                    xCraneAtHome
                    OR (
                        xMotionStarted
                        AND NOT xMovingX
                        AND NOT xMovingZ
                    )
                )
            THEN
                xMotionStarted := FALSE;

                IF xDepositComplete THEN
                    eState := E_StorageState.Complete;
                ELSE
                    eState := E_StorageState.Idle;
                END_IF;
            END_IF;


        E_StorageState.Complete:
            wTargetPositionCmd := wHomePosition;

            // Hold completion until Batch Storage removes its request.
            IF NOT xStoreRequest THEN
                wActivePosition := 0;
                xDepositComplete := FALSE;
                eState := E_StorageState.Idle;
            END_IF;


        E_StorageState.Faulted:
            // Boolean outputs remain at their safe defaults.


    ELSE
        uiFaultCode := 799;
        xReservationFault := TRUE;
        eState := E_StorageState.Faulted;

    END_CASE;
END_IF;

// Only active physical steps use the common progress timeout.
xTimedStep :=
    (eState = E_StorageState.ReceivingProduct)
    OR (eState = E_StorageState.ExtendingToLoad)
    OR (eState = E_StorageState.LiftingProduct)
    OR (eState = E_StorageState.RetractingWithProduct)
    OR (eState = E_StorageState.MovingToRack)
    OR (eState = E_StorageState.ExtendingToRack)
    OR (eState = E_StorageState.LoweringProduct)
    OR (eState = E_StorageState.RetractingAfterDeposit)
    OR (eState = E_StorageState.ReturningHome);

xStateChanged := eState <> ePreviousState;

fbStepTimeout(
    IN :=
        xEnable
        AND xRun
        AND xTimedStep
        AND NOT xStateChanged,
    PT := tStepTimeout
);

ePreviousState := eState;

IF fbStepTimeout.Q THEN
    uiFaultCode := 711;
    xStepTimeoutFault := TRUE;
END_IF;

xFaulted :=
    xReservationFault
    OR xStepTimeoutFault;

// Remove commands immediately when a fault is discovered.
IF xFaulted THEN
    eState := E_StorageState.Faulted;
    xCommandArmed := FALSE;
    xEntryConveyorCmd := FALSE;
    xForksLeftCmd := FALSE;
    xForksRightCmd := FALSE;
    xLiftCmd := FALSE;
    xLoadConveyorCmd := FALSE;
END_IF;

// Public status.
xBusy :=
    (eState <> E_StorageState.Stopped)
    AND (eState <> E_StorageState.Idle)
    AND (eState <> E_StorageState.Complete)
    AND (eState <> E_StorageState.Faulted);

xReady :=
    xEnable
    AND xRun
    AND NOT xFaulted
    AND (eState = E_StorageState.Idle);

xStoreComplete :=
    NOT xFaulted
    AND (eState = E_StorageState.Complete);

END_FUNCTION_BLOCK

